// TIA Portal V17 export
// export: Created 2024-09-02T12:50:08.8547396Z, ExportSetting WithDefaults, DisplayName Totally Integrated Automation Portal, DisplayVersion V17, DisplayName TIA Portal Openness, DisplayVersion V17, DisplayName TIA Portal Version Control Interface, DisplayVersion V17, DisplayName STEP 7 Professional, DisplayVersion V17, DisplayName STEP 7 Safety, DisplayVersion V17, DisplayName WinCC Professional, DisplayVersion V17
FUNCTION "AnwFC2_FG02_Station_OP70" : Void   // FC1382, LAD
TITLE = Station
{ S7_Optimized_Access := 'TRUE' }
AUTHOR : VAF
FAMILY : SK
NAME : SK
VERSION : 0.1
// stored: AutoNumber false, IsIECCheckEnabled false, SetENOAutomatically false, UDAEnableTagReadback false
   VAR_TEMP
      Motion_Release : Bool;   // Motion permit
      Hand : Bool;
      Auto : Bool;
      t_Ret_Val_SFC : Int;
      t_fm_Gen : Bool;
      t_ParityFault : Bool;
      t_ConfigFault : Bool;
      t_Retval : Bool;
      MM150_Work : Bool;
      MM150_Home : Bool;
      MM160_Work : Bool;
      MM160_Home : Bool;
      MM170_Work : Bool;
      MM170_Home : Bool;
      MM140_Home : Bool;
      MM140_Work : Bool;
      X1 : Int;
      X2 : Int;
      Y : Int;
      X_actual : Int;
      dummy : Bool;
   END_VAR
   VAR_TEMP   // added for the SCL form of the ladder/FBD networks
      _w1 : Bool;
      _w2 : Bool;
   END_VAR
BEGIN

REGION Network 1: Motion permit / Hand/ Auto
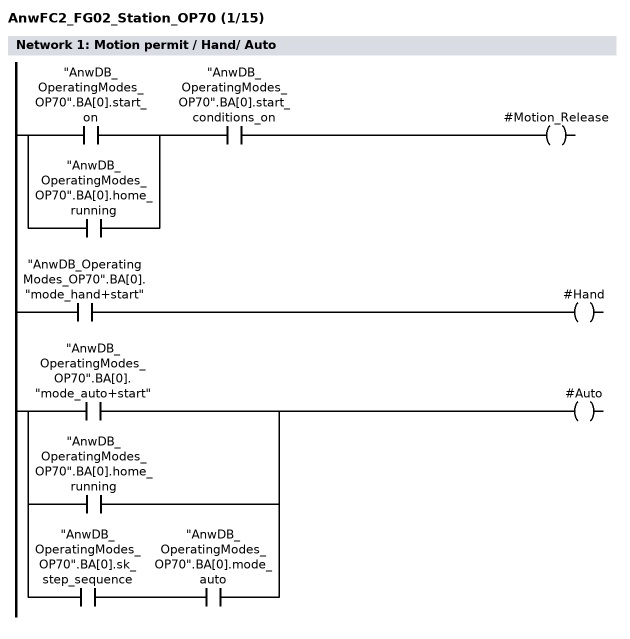
   RUNG wire#powerrail
      Contact( "AnwDB_OperatingModes_OP70".BA[0].start_on )
      wire#w1
      Contact( "AnwDB_OperatingModes_OP70".BA[0].start_conditions_on )
      Coil( #Motion_Release )
   END_RUNG
   RUNG wire#powerrail
      Contact( "AnwDB_OperatingModes_OP70".BA[0].home_running )
   END_RUNG wire#w1
   RUNG wire#powerrail
      Contact( "AnwDB_OperatingModes_OP70".BA[0]."mode_hand+start" )
      Coil( #Hand )
   END_RUNG
   RUNG wire#powerrail
      Contact( "AnwDB_OperatingModes_OP70".BA[0]."mode_auto+start" )
      wire#w2
      Coil( #Auto )
   END_RUNG
   RUNG wire#powerrail
      Contact( "AnwDB_OperatingModes_OP70".BA[0].home_running )
   END_RUNG wire#w2
   RUNG wire#powerrail
      Contact( "AnwDB_OperatingModes_OP70".BA[0].sk_step_sequence )
      Contact( "AnwDB_OperatingModes_OP70".BA[0].mode_auto )
   END_RUNG wire#w2
   // the same network as SCL:
   #Motion_Release := ("AnwDB_OperatingModes_OP70".BA[0].start_on OR "AnwDB_OperatingModes_OP70".BA[0].home_running) AND "AnwDB_OperatingModes_OP70".BA[0].start_conditions_on;
   #Hand := "AnwDB_OperatingModes_OP70".BA[0]."mode_hand+start";
   #Auto := "AnwDB_OperatingModes_OP70".BA[0]."mode_auto+start" OR "AnwDB_OperatingModes_OP70".BA[0].home_running OR ("AnwDB_OperatingModes_OP70".BA[0].sk_step_sequence AND "AnwDB_OperatingModes_OP70".BA[0].mode_auto);
END_REGION

REGION Network 2: Call of the step sequence
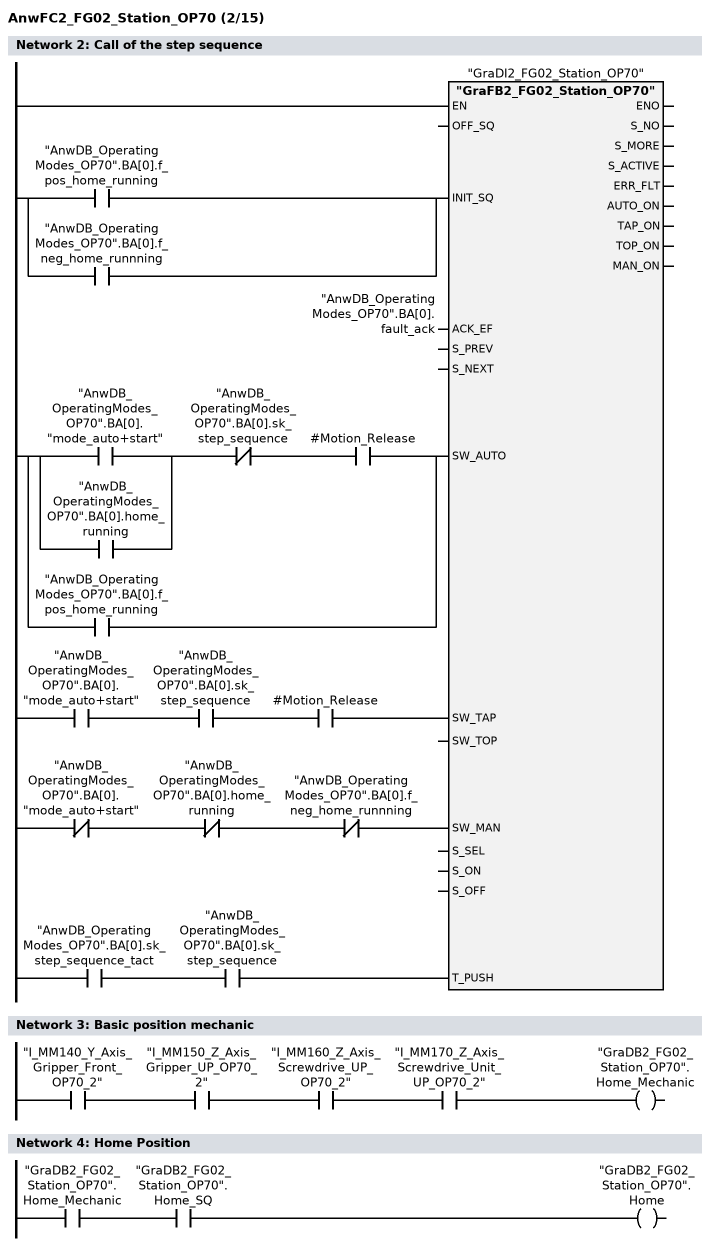
   RUNG wire#powerrail
      "GraDI2_FG02_Station_OP70"(INIT_SQ := wire#w1, SW_AUTO := wire#w3, SW_TAP := wire#w4, SW_MAN := wire#w5, T_PUSH := wire#w6, OFF_SQ :=, ACK_EF := "AnwDB_OperatingModes_OP70".BA[0].fault_ack, S_PREV :=, S_NEXT :=, SW_TOP :=, S_SEL :=, S_ON :=, S_OFF :=, S_NO =>, S_MORE =>, S_ACTIVE =>, ERR_FLT =>, AUTO_ON =>, TAP_ON =>, TOP_ON =>, MAN_ON =>)
   END_RUNG
   RUNG wire#powerrail
      Contact( "AnwDB_OperatingModes_OP70".BA[0].f_pos_home_running )
   END_RUNG wire#w1
   RUNG wire#powerrail
      Contact( "AnwDB_OperatingModes_OP70".BA[0].f_neg_home_runnning )
   END_RUNG wire#w1
   RUNG wire#powerrail
      Contact( "AnwDB_OperatingModes_OP70".BA[0]."mode_auto+start" )
      wire#w2
      I_Contact( "AnwDB_OperatingModes_OP70".BA[0].sk_step_sequence )
      Contact( #Motion_Release )
   END_RUNG wire#w3
   RUNG wire#powerrail
      Contact( "AnwDB_OperatingModes_OP70".BA[0].home_running )
   END_RUNG wire#w2
   RUNG wire#powerrail
      Contact( "AnwDB_OperatingModes_OP70".BA[0].f_pos_home_running )
   END_RUNG wire#w3
   RUNG wire#powerrail
      Contact( "AnwDB_OperatingModes_OP70".BA[0]."mode_auto+start" )
      Contact( "AnwDB_OperatingModes_OP70".BA[0].sk_step_sequence )
      Contact( #Motion_Release )
   END_RUNG wire#w4
   RUNG wire#powerrail
      I_Contact( "AnwDB_OperatingModes_OP70".BA[0]."mode_auto+start" )
      I_Contact( "AnwDB_OperatingModes_OP70".BA[0].home_running )
      I_Contact( "AnwDB_OperatingModes_OP70".BA[0].f_neg_home_runnning )
   END_RUNG wire#w5
   RUNG wire#powerrail
      Contact( "AnwDB_OperatingModes_OP70".BA[0].sk_step_sequence_tact )
      Contact( "AnwDB_OperatingModes_OP70".BA[0].sk_step_sequence )
   END_RUNG wire#w6
   // the same network as SCL:
   "GraDI2_FG02_Station_OP70"(INIT_SQ := "AnwDB_OperatingModes_OP70".BA[0].f_pos_home_running OR "AnwDB_OperatingModes_OP70".BA[0].f_neg_home_runnning,   // "GraFB2_FG02_Station_OP70"
                           ACK_EF := "AnwDB_OperatingModes_OP70".BA[0].fault_ack,
                           SW_AUTO := (("AnwDB_OperatingModes_OP70".BA[0]."mode_auto+start" OR "AnwDB_OperatingModes_OP70".BA[0].home_running) AND NOT "AnwDB_OperatingModes_OP70".BA[0].sk_step_sequence AND #Motion_Release) OR "AnwDB_OperatingModes_OP70".BA[0].f_pos_home_running,
                           SW_TAP := "AnwDB_OperatingModes_OP70".BA[0]."mode_auto+start" AND "AnwDB_OperatingModes_OP70".BA[0].sk_step_sequence AND #Motion_Release,
                           SW_MAN := NOT "AnwDB_OperatingModes_OP70".BA[0]."mode_auto+start" AND NOT "AnwDB_OperatingModes_OP70".BA[0].home_running AND NOT "AnwDB_OperatingModes_OP70".BA[0].f_neg_home_runnning,
                           T_PUSH := "AnwDB_OperatingModes_OP70".BA[0].sk_step_sequence_tact AND "AnwDB_OperatingModes_OP70".BA[0].sk_step_sequence);
END_REGION

REGION Network 3: Basic position mechanic
   RUNG wire#powerrail
      Contact( "I_MM140_Y_Axis_Gripper_Front_OP70_2" )
      Contact( "I_MM150_Z_Axis_Gripper_UP_OP70_2" )
      Contact( "I_MM160_Z_Axis_Screwdrive_UP_OP70_2" )
      Contact( "I_MM170_Z_Axis_Screwdrive_Unit_UP_OP70_2" )
      Coil( "GraDB2_FG02_Station_OP70".Home_Mechanic )
   END_RUNG
   // the same network as SCL:
   "GraDB2_FG02_Station_OP70".Home_Mechanic := "I_MM140_Y_Axis_Gripper_Front_OP70_2" AND "I_MM150_Z_Axis_Gripper_UP_OP70_2" AND "I_MM160_Z_Axis_Screwdrive_UP_OP70_2" AND "I_MM170_Z_Axis_Screwdrive_Unit_UP_OP70_2";
END_REGION

REGION Network 4: Home Position
   RUNG wire#powerrail
      Contact( "GraDB2_FG02_Station_OP70".Home_Mechanic )
      Contact( "GraDB2_FG02_Station_OP70".Home_SQ )
      Coil( "GraDB2_FG02_Station_OP70".Home )
   END_RUNG
   // the same network as SCL:
   "GraDB2_FG02_Station_OP70".Home := "GraDB2_FG02_Station_OP70".Home_Mechanic AND "GraDB2_FG02_Station_OP70".Home_SQ;
END_REGION

REGION Network 5: ########### USER ###########
END_REGION

REGION Network 6: Screen selection with NOK BEA1
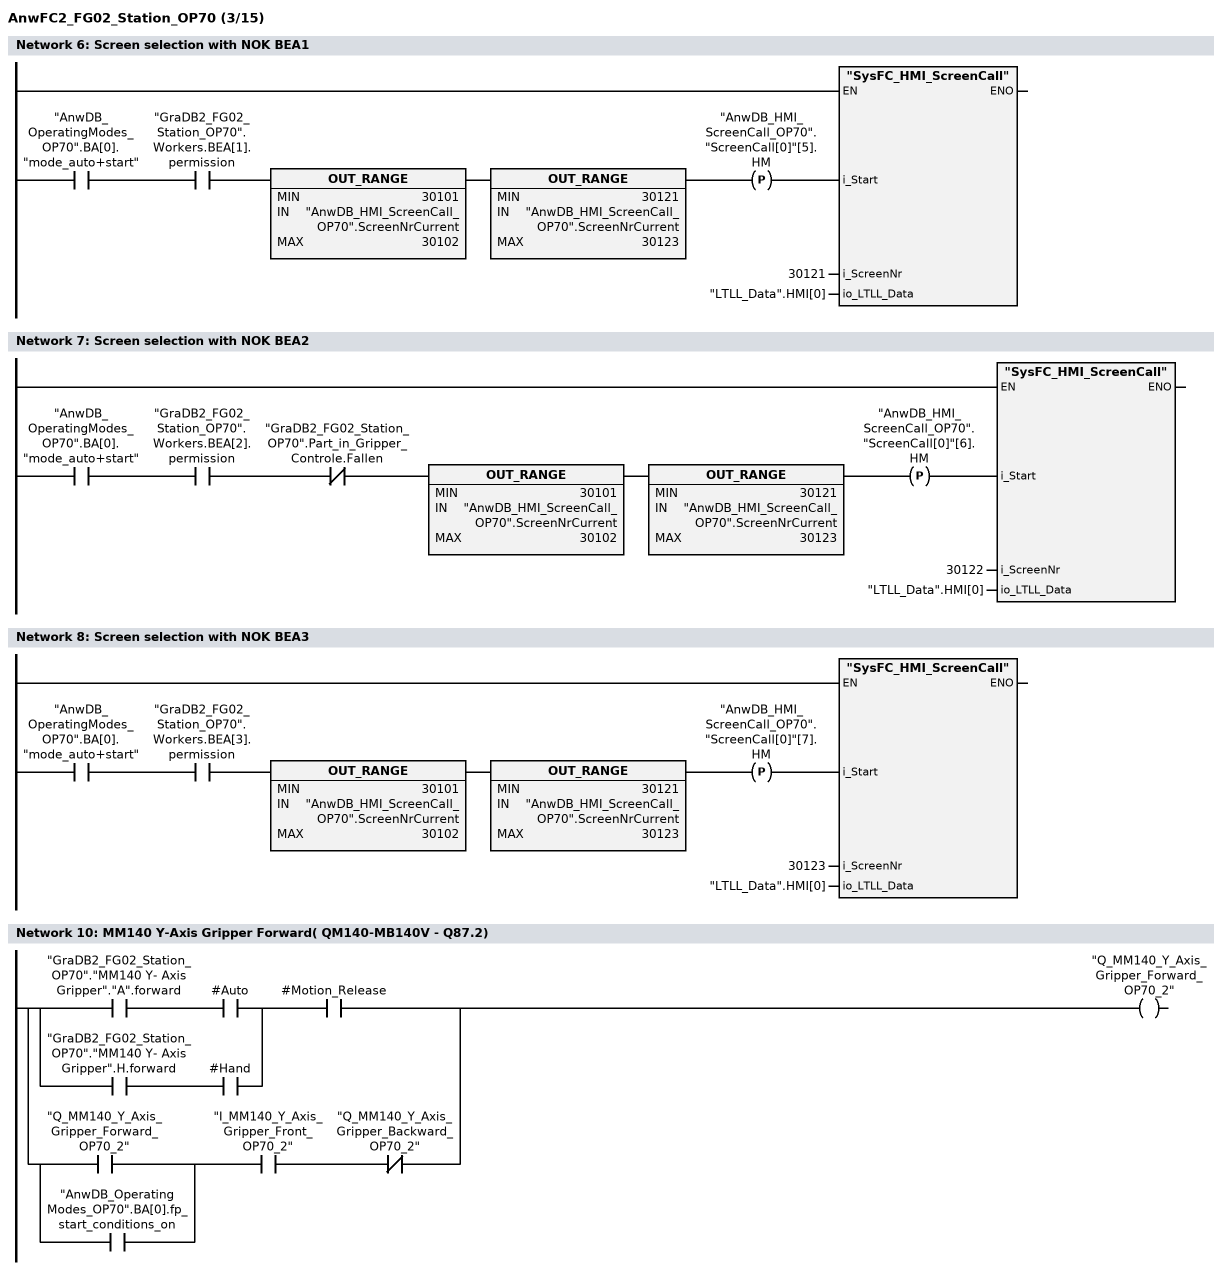
   #_w1 := "AnwDB_OperatingModes_OP70".BA[0]."mode_auto+start" AND "GraDB2_FG02_Station_OP70".Workers.BEA[1].permission AND (("AnwDB_HMI_ScreenCall_OP70".ScreenNrCurrent < 30101) OR ("AnwDB_HMI_ScreenCall_OP70".ScreenNrCurrent > 30102)) AND (("AnwDB_HMI_ScreenCall_OP70".ScreenNrCurrent < 30121) OR ("AnwDB_HMI_ScreenCall_OP70".ScreenNrCurrent > 30123));
   #_w2 := #_w1 AND NOT "AnwDB_HMI_ScreenCall_OP70"."ScreenCall[0]"[5].HM;   // rising edge
   "AnwDB_HMI_ScreenCall_OP70"."ScreenCall[0]"[5].HM := #_w1;
   "SysFC_HMI_ScreenCall"(i_Start := #_w2, i_ScreenNr := 30121, io_LTLL_Data := "LTLL_Data".HMI[0]);
END_REGION

REGION Network 7: Screen selection with NOK BEA2
   #_w1 := "AnwDB_OperatingModes_OP70".BA[0]."mode_auto+start" AND "GraDB2_FG02_Station_OP70".Workers.BEA[2].permission AND NOT "GraDB2_FG02_Station_OP70".Part_in_Gripper_Controle.Fallen AND (("AnwDB_HMI_ScreenCall_OP70".ScreenNrCurrent < 30101) OR ("AnwDB_HMI_ScreenCall_OP70".ScreenNrCurrent > 30102)) AND (("AnwDB_HMI_ScreenCall_OP70".ScreenNrCurrent < 30121) OR ("AnwDB_HMI_ScreenCall_OP70".ScreenNrCurrent > 30123));
   #_w2 := #_w1 AND NOT "AnwDB_HMI_ScreenCall_OP70"."ScreenCall[0]"[6].HM;   // rising edge
   "AnwDB_HMI_ScreenCall_OP70"."ScreenCall[0]"[6].HM := #_w1;
   "SysFC_HMI_ScreenCall"(i_Start := #_w2, i_ScreenNr := 30122, io_LTLL_Data := "LTLL_Data".HMI[0]);
END_REGION

REGION Network 8: Screen selection with NOK BEA3
   #_w1 := "AnwDB_OperatingModes_OP70".BA[0]."mode_auto+start" AND "GraDB2_FG02_Station_OP70".Workers.BEA[3].permission AND (("AnwDB_HMI_ScreenCall_OP70".ScreenNrCurrent < 30101) OR ("AnwDB_HMI_ScreenCall_OP70".ScreenNrCurrent > 30102)) AND (("AnwDB_HMI_ScreenCall_OP70".ScreenNrCurrent < 30121) OR ("AnwDB_HMI_ScreenCall_OP70".ScreenNrCurrent > 30123));
   #_w2 := #_w1 AND NOT "AnwDB_HMI_ScreenCall_OP70"."ScreenCall[0]"[7].HM;   // rising edge
   "AnwDB_HMI_ScreenCall_OP70"."ScreenCall[0]"[7].HM := #_w1;
   "SysFC_HMI_ScreenCall"(i_Start := #_w2, i_ScreenNr := 30123, io_LTLL_Data := "LTLL_Data".HMI[0]);
END_REGION

REGION Network 9: ########### SS_02_001_Setup ###########
END_REGION

REGION Network 10: MM140 Y-Axis Gripper Forward( QM140-MB140V - Q87.2)
   RUNG wire#powerrail
      Contact( "GraDB2_FG02_Station_OP70"."MM140 Y- Axis Gripper"."A".forward )
      Contact( #Auto )
      wire#w1
      Contact( #Motion_Release )
      wire#w2
      Coil( "Q_MM140_Y_Axis_Gripper_Forward_OP70_2" )
   END_RUNG
   RUNG wire#powerrail
      Contact( "GraDB2_FG02_Station_OP70"."MM140 Y- Axis Gripper".H.forward )
      Contact( #Hand )
   END_RUNG wire#w1
   RUNG wire#powerrail
      Contact( "Q_MM140_Y_Axis_Gripper_Forward_OP70_2" )
      wire#w3
      Contact( "I_MM140_Y_Axis_Gripper_Front_OP70_2" )
      I_Contact( "Q_MM140_Y_Axis_Gripper_Backward_OP70_2" )
   END_RUNG wire#w2
   RUNG wire#powerrail
      Contact( "AnwDB_OperatingModes_OP70".BA[0].fp_start_conditions_on )
   END_RUNG wire#w3
   // the same network as SCL:
   "Q_MM140_Y_Axis_Gripper_Forward_OP70_2" := ((("GraDB2_FG02_Station_OP70"."MM140 Y- Axis Gripper"."A".forward AND #Auto) OR ("GraDB2_FG02_Station_OP70"."MM140 Y- Axis Gripper".H.forward AND #Hand)) AND #Motion_Release) OR (("Q_MM140_Y_Axis_Gripper_Forward_OP70_2" OR "AnwDB_OperatingModes_OP70".BA[0].fp_start_conditions_on) AND "I_MM140_Y_Axis_Gripper_Front_OP70_2" AND NOT "Q_MM140_Y_Axis_Gripper_Backward_OP70_2");
END_REGION

REGION Network 11: MM140 Y-Axis Gripper Backward( QM140-MB140R - Q87.3 )
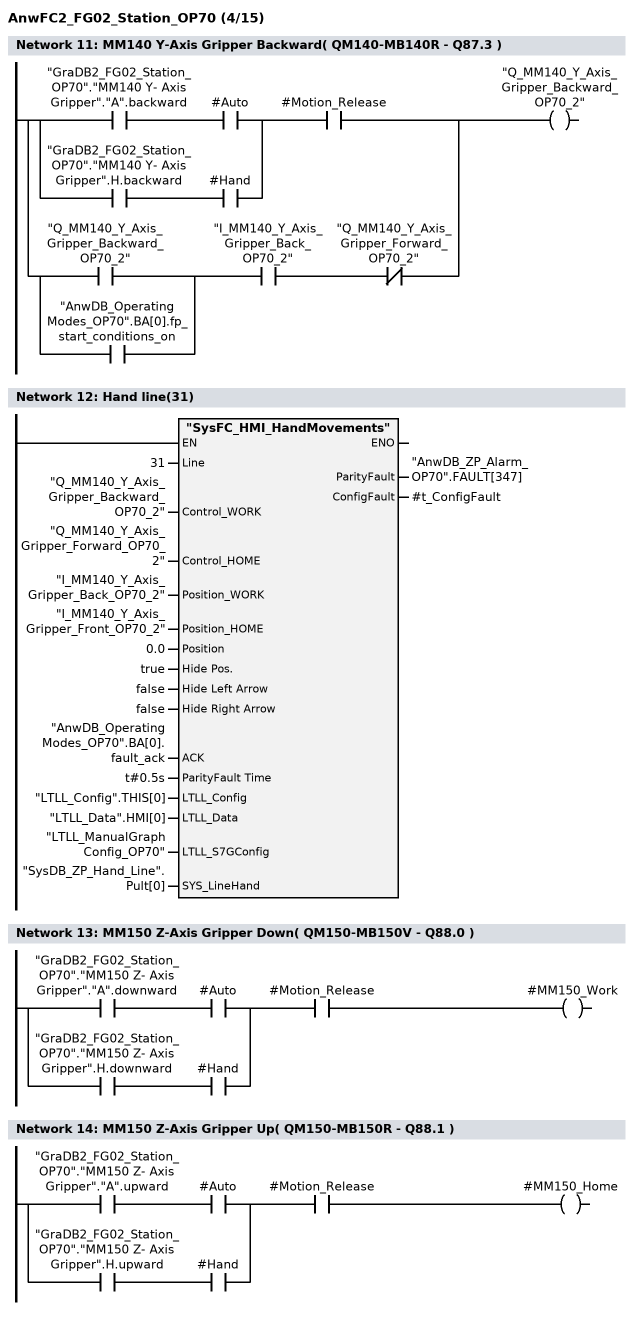
   RUNG wire#powerrail
      Contact( "GraDB2_FG02_Station_OP70"."MM140 Y- Axis Gripper"."A".backward )
      Contact( #Auto )
      wire#w1
      Contact( #Motion_Release )
      wire#w2
      Coil( "Q_MM140_Y_Axis_Gripper_Backward_OP70_2" )
   END_RUNG
   RUNG wire#powerrail
      Contact( "GraDB2_FG02_Station_OP70"."MM140 Y- Axis Gripper".H.backward )
      Contact( #Hand )
   END_RUNG wire#w1
   RUNG wire#powerrail
      Contact( "Q_MM140_Y_Axis_Gripper_Backward_OP70_2" )
      wire#w3
      Contact( "I_MM140_Y_Axis_Gripper_Back_OP70_2" )
      I_Contact( "Q_MM140_Y_Axis_Gripper_Forward_OP70_2" )
   END_RUNG wire#w2
   RUNG wire#powerrail
      Contact( "AnwDB_OperatingModes_OP70".BA[0].fp_start_conditions_on )
   END_RUNG wire#w3
   // the same network as SCL:
   "Q_MM140_Y_Axis_Gripper_Backward_OP70_2" := ((("GraDB2_FG02_Station_OP70"."MM140 Y- Axis Gripper"."A".backward AND #Auto) OR ("GraDB2_FG02_Station_OP70"."MM140 Y- Axis Gripper".H.backward AND #Hand)) AND #Motion_Release) OR (("Q_MM140_Y_Axis_Gripper_Backward_OP70_2" OR "AnwDB_OperatingModes_OP70".BA[0].fp_start_conditions_on) AND "I_MM140_Y_Axis_Gripper_Back_OP70_2" AND NOT "Q_MM140_Y_Axis_Gripper_Forward_OP70_2");
END_REGION

REGION Network 12: Hand line(31)
   RUNG wire#powerrail
      "SysFC_HMI_HandMovements"(Line := 31, Control_WORK := "Q_MM140_Y_Axis_Gripper_Backward_OP70_2", Control_HOME := "Q_MM140_Y_Axis_Gripper_Forward_OP70_2", Position_WORK := "I_MM140_Y_Axis_Gripper_Back_OP70_2", Position_HOME := "I_MM140_Y_Axis_Gripper_Front_OP70_2", Position := 0.0, "Hide Pos." := true, "Hide Left Arrow" := false, "Hide Right Arrow" := false, ACK := "AnwDB_OperatingModes_OP70".BA[0].fault_ack, "ParityFault Time" := t#0.5s, LTLL_Config := "LTLL_Config".THIS[0], LTLL_Data := "LTLL_Data".HMI[0], LTLL_S7GConfig := "LTLL_ManualGraphConfig_OP70", SYS_LineHand := "SysDB_ZP_Hand_Line".Pult[0], ParityFault => "AnwDB_ZP_Alarm_OP70".FAULT[347], ConfigFault => #t_ConfigFault)
   END_RUNG
   // the same network as SCL:
   "SysFC_HMI_HandMovements"(Line := 31,
                           Control_WORK := "Q_MM140_Y_Axis_Gripper_Backward_OP70_2",
                           Control_HOME := "Q_MM140_Y_Axis_Gripper_Forward_OP70_2",
                           Position_WORK := "I_MM140_Y_Axis_Gripper_Back_OP70_2",
                           Position_HOME := "I_MM140_Y_Axis_Gripper_Front_OP70_2",
                           Position := 0.0,
                           "Hide Pos." := true,
                           "Hide Left Arrow" := false,
                           "Hide Right Arrow" := false,
                           ACK := "AnwDB_OperatingModes_OP70".BA[0].fault_ack,
                           "ParityFault Time" := t#0.5s,
                           LTLL_Config := "LTLL_Config".THIS[0],
                           LTLL_Data := "LTLL_Data".HMI[0],
                           LTLL_S7GConfig := "LTLL_ManualGraphConfig_OP70",
                           SYS_LineHand := "SysDB_ZP_Hand_Line".Pult[0],
                           ParityFault => "AnwDB_ZP_Alarm_OP70".FAULT[347],
                           ConfigFault => #t_ConfigFault);
END_REGION

REGION Network 13: MM150 Z-Axis Gripper Down( QM150-MB150V - Q88.0 )
   RUNG wire#powerrail
      Contact( "GraDB2_FG02_Station_OP70"."MM150 Z- Axis Gripper"."A".downward )
      Contact( #Auto )
      wire#w1
      Contact( #Motion_Release )
      Coil( #MM150_Work )
   END_RUNG
   RUNG wire#powerrail
      Contact( "GraDB2_FG02_Station_OP70"."MM150 Z- Axis Gripper".H.downward )
      Contact( #Hand )
   END_RUNG wire#w1
   // the same network as SCL:
   #MM150_Work := (("GraDB2_FG02_Station_OP70"."MM150 Z- Axis Gripper"."A".downward AND #Auto) OR ("GraDB2_FG02_Station_OP70"."MM150 Z- Axis Gripper".H.downward AND #Hand)) AND #Motion_Release;
END_REGION

REGION Network 14: MM150 Z-Axis Gripper Up( QM150-MB150R - Q88.1 )
   RUNG wire#powerrail
      Contact( "GraDB2_FG02_Station_OP70"."MM150 Z- Axis Gripper"."A".upward )
      Contact( #Auto )
      wire#w1
      Contact( #Motion_Release )
      Coil( #MM150_Home )
   END_RUNG
   RUNG wire#powerrail
      Contact( "GraDB2_FG02_Station_OP70"."MM150 Z- Axis Gripper".H.upward )
      Contact( #Hand )
   END_RUNG wire#w1
   // the same network as SCL:
   #MM150_Home := (("GraDB2_FG02_Station_OP70"."MM150 Z- Axis Gripper"."A".upward AND #Auto) OR ("GraDB2_FG02_Station_OP70"."MM150 Z- Axis Gripper".H.upward AND #Hand)) AND #Motion_Release;
END_REGION

REGION Network 15: HLP - Z-Axis Gripper Up/Down
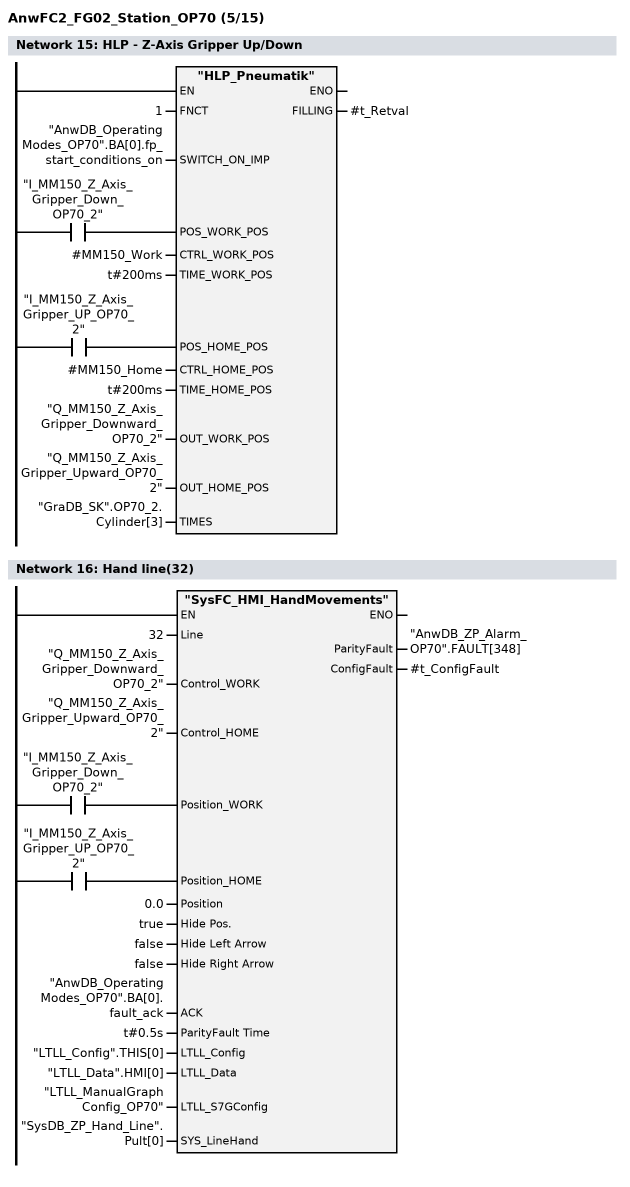
   RUNG wire#powerrail
      "HLP_Pneumatik"(POS_WORK_POS := wire#w1, POS_HOME_POS := wire#w2, FNCT := 1, SWITCH_ON_IMP := "AnwDB_OperatingModes_OP70".BA[0].fp_start_conditions_on, CTRL_WORK_POS := #MM150_Work, TIME_WORK_POS := t#200ms, CTRL_HOME_POS := #MM150_Home, TIME_HOME_POS := t#200ms, OUT_WORK_POS := "Q_MM150_Z_Axis_Gripper_Downward_OP70_2", OUT_HOME_POS := "Q_MM150_Z_Axis_Gripper_Upward_OP70_2", TIMES := "GraDB_SK".OP70_2.Cylinder[3], FILLING => #t_Retval)
   END_RUNG
   RUNG wire#powerrail
      Contact( "I_MM150_Z_Axis_Gripper_Down_OP70_2" )
   END_RUNG wire#w1
   RUNG wire#powerrail
      Contact( "I_MM150_Z_Axis_Gripper_UP_OP70_2" )
   END_RUNG wire#w2
   // the same network as SCL:
   "HLP_Pneumatik"(FNCT := 1,
                   SWITCH_ON_IMP := "AnwDB_OperatingModes_OP70".BA[0].fp_start_conditions_on,
                   POS_WORK_POS := "I_MM150_Z_Axis_Gripper_Down_OP70_2",
                   CTRL_WORK_POS := #MM150_Work,
                   TIME_WORK_POS := t#200ms,
                   POS_HOME_POS := "I_MM150_Z_Axis_Gripper_UP_OP70_2",
                   CTRL_HOME_POS := #MM150_Home,
                   TIME_HOME_POS := t#200ms,
                   OUT_WORK_POS := "Q_MM150_Z_Axis_Gripper_Downward_OP70_2",
                   OUT_HOME_POS := "Q_MM150_Z_Axis_Gripper_Upward_OP70_2",
                   TIMES := "GraDB_SK".OP70_2.Cylinder[3],
                   FILLING => #t_Retval);
END_REGION

REGION Network 16: Hand line(32)
   RUNG wire#powerrail
      "SysFC_HMI_HandMovements"(Position_WORK := wire#w1, Position_HOME := wire#w2, Line := 32, Control_WORK := "Q_MM150_Z_Axis_Gripper_Downward_OP70_2", Control_HOME := "Q_MM150_Z_Axis_Gripper_Upward_OP70_2", Position := 0.0, "Hide Pos." := true, "Hide Left Arrow" := false, "Hide Right Arrow" := false, ACK := "AnwDB_OperatingModes_OP70".BA[0].fault_ack, "ParityFault Time" := t#0.5s, LTLL_Config := "LTLL_Config".THIS[0], LTLL_Data := "LTLL_Data".HMI[0], LTLL_S7GConfig := "LTLL_ManualGraphConfig_OP70", SYS_LineHand := "SysDB_ZP_Hand_Line".Pult[0], ParityFault => "AnwDB_ZP_Alarm_OP70".FAULT[348], ConfigFault => #t_ConfigFault)
   END_RUNG
   RUNG wire#powerrail
      Contact( "I_MM150_Z_Axis_Gripper_Down_OP70_2" )
   END_RUNG wire#w1
   RUNG wire#powerrail
      Contact( "I_MM150_Z_Axis_Gripper_UP_OP70_2" )
   END_RUNG wire#w2
   // the same network as SCL:
   "SysFC_HMI_HandMovements"(Line := 32,
                           Control_WORK := "Q_MM150_Z_Axis_Gripper_Downward_OP70_2",
                           Control_HOME := "Q_MM150_Z_Axis_Gripper_Upward_OP70_2",
                           Position_WORK := "I_MM150_Z_Axis_Gripper_Down_OP70_2",
                           Position_HOME := "I_MM150_Z_Axis_Gripper_UP_OP70_2",
                           Position := 0.0,
                           "Hide Pos." := true,
                           "Hide Left Arrow" := false,
                           "Hide Right Arrow" := false,
                           ACK := "AnwDB_OperatingModes_OP70".BA[0].fault_ack,
                           "ParityFault Time" := t#0.5s,
                           LTLL_Config := "LTLL_Config".THIS[0],
                           LTLL_Data := "LTLL_Data".HMI[0],
                           LTLL_S7GConfig := "LTLL_ManualGraphConfig_OP70",
                           SYS_LineHand := "SysDB_ZP_Hand_Line".Pult[0],
                           ParityFault => "AnwDB_ZP_Alarm_OP70".FAULT[348],
                           ConfigFault => #t_ConfigFault);
END_REGION

REGION Network 17: Voccum Gripper Open ######( QM303-MBXXXR - Q2.1)
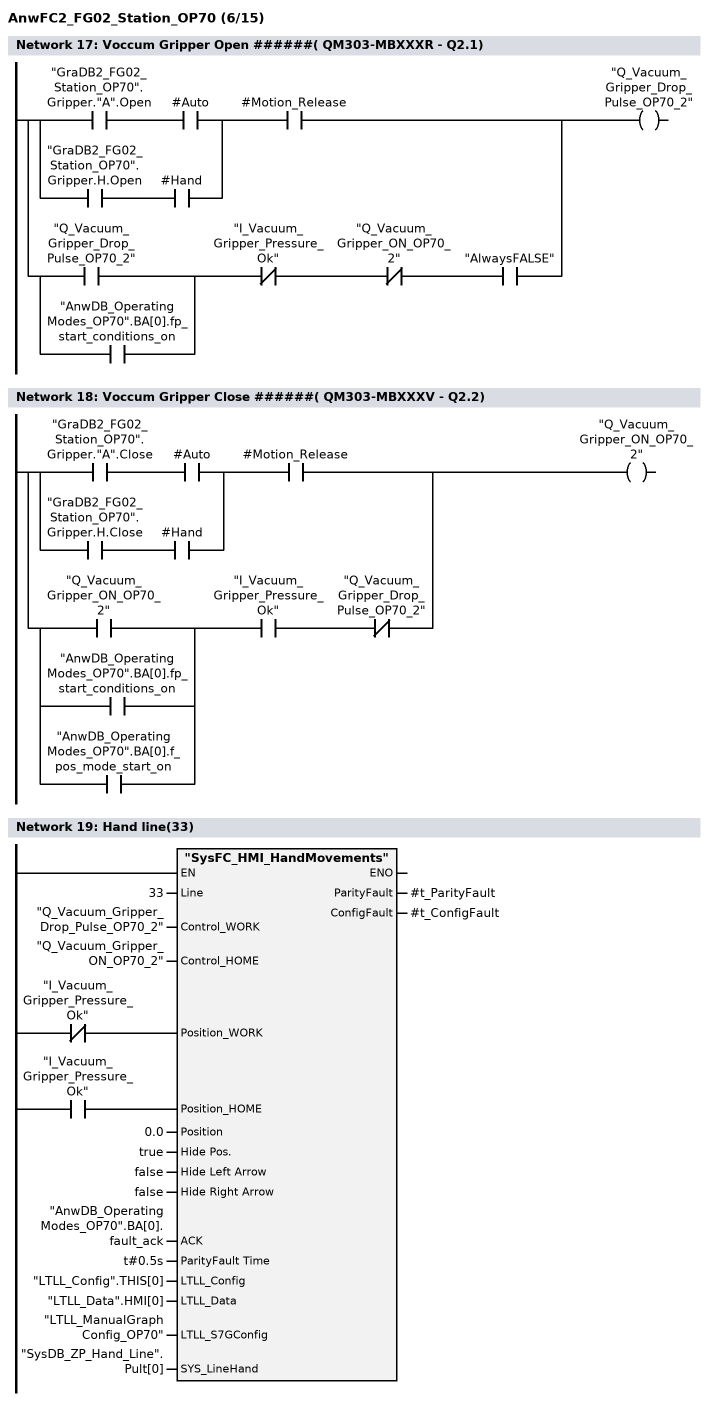
   RUNG wire#powerrail
      Contact( "GraDB2_FG02_Station_OP70".Gripper."A".Open )
      Contact( #Auto )
      wire#w1
      Contact( #Motion_Release )
      wire#w2
      Coil( "Q_Vacuum_Gripper_Drop_Pulse_OP70_2" )
   END_RUNG
   RUNG wire#powerrail
      Contact( "GraDB2_FG02_Station_OP70".Gripper.H.Open )
      Contact( #Hand )
   END_RUNG wire#w1
   RUNG wire#powerrail
      Contact( "Q_Vacuum_Gripper_Drop_Pulse_OP70_2" )
      wire#w3
      I_Contact( "I_Vacuum_Gripper_Pressure_Ok" )
      I_Contact( "Q_Vacuum_Gripper_ON_OP70_2" )
      Contact( "AlwaysFALSE" )
   END_RUNG wire#w2
   RUNG wire#powerrail
      Contact( "AnwDB_OperatingModes_OP70".BA[0].fp_start_conditions_on )
   END_RUNG wire#w3
   // the same network as SCL:
   "Q_Vacuum_Gripper_Drop_Pulse_OP70_2" := ((("GraDB2_FG02_Station_OP70".Gripper."A".Open AND #Auto) OR ("GraDB2_FG02_Station_OP70".Gripper.H.Open AND #Hand)) AND #Motion_Release) OR (("Q_Vacuum_Gripper_Drop_Pulse_OP70_2" OR "AnwDB_OperatingModes_OP70".BA[0].fp_start_conditions_on) AND NOT "I_Vacuum_Gripper_Pressure_Ok" AND NOT "Q_Vacuum_Gripper_ON_OP70_2" AND "AlwaysFALSE");
END_REGION

REGION Network 18: Voccum Gripper Close ######( QM303-MBXXXV - Q2.2)
   RUNG wire#powerrail
      Contact( "GraDB2_FG02_Station_OP70".Gripper."A".Close )
      Contact( #Auto )
      wire#w1
      Contact( #Motion_Release )
      wire#w2
      Coil( "Q_Vacuum_Gripper_ON_OP70_2" )
   END_RUNG
   RUNG wire#powerrail
      Contact( "GraDB2_FG02_Station_OP70".Gripper.H.Close )
      Contact( #Hand )
   END_RUNG wire#w1
   RUNG wire#powerrail
      Contact( "Q_Vacuum_Gripper_ON_OP70_2" )
      wire#w3
      Contact( "I_Vacuum_Gripper_Pressure_Ok" )
      I_Contact( "Q_Vacuum_Gripper_Drop_Pulse_OP70_2" )
   END_RUNG wire#w2
   RUNG wire#powerrail
      Contact( "AnwDB_OperatingModes_OP70".BA[0].fp_start_conditions_on )
   END_RUNG wire#w3
   RUNG wire#powerrail
      Contact( "AnwDB_OperatingModes_OP70".BA[0].f_pos_mode_start_on )
   END_RUNG wire#w3
   // the same network as SCL:
   "Q_Vacuum_Gripper_ON_OP70_2" := ((("GraDB2_FG02_Station_OP70".Gripper."A".Close AND #Auto) OR ("GraDB2_FG02_Station_OP70".Gripper.H.Close AND #Hand)) AND #Motion_Release) OR (("Q_Vacuum_Gripper_ON_OP70_2" OR "AnwDB_OperatingModes_OP70".BA[0].fp_start_conditions_on OR "AnwDB_OperatingModes_OP70".BA[0].f_pos_mode_start_on) AND "I_Vacuum_Gripper_Pressure_Ok" AND NOT "Q_Vacuum_Gripper_Drop_Pulse_OP70_2");
END_REGION

REGION Network 19: Hand line(33)
   RUNG wire#powerrail
      "SysFC_HMI_HandMovements"(Position_WORK := wire#w1, Position_HOME := wire#w2, Line := 33, Control_WORK := "Q_Vacuum_Gripper_Drop_Pulse_OP70_2", Control_HOME := "Q_Vacuum_Gripper_ON_OP70_2", Position := 0.0, "Hide Pos." := true, "Hide Left Arrow" := false, "Hide Right Arrow" := false, ACK := "AnwDB_OperatingModes_OP70".BA[0].fault_ack, "ParityFault Time" := t#0.5s, LTLL_Config := "LTLL_Config".THIS[0], LTLL_Data := "LTLL_Data".HMI[0], LTLL_S7GConfig := "LTLL_ManualGraphConfig_OP70", SYS_LineHand := "SysDB_ZP_Hand_Line".Pult[0], ParityFault => #t_ParityFault, ConfigFault => #t_ConfigFault)
   END_RUNG
   RUNG wire#powerrail
      I_Contact( "I_Vacuum_Gripper_Pressure_Ok" )
   END_RUNG wire#w1
   RUNG wire#powerrail
      Contact( "I_Vacuum_Gripper_Pressure_Ok" )
   END_RUNG wire#w2
   // the same network as SCL:
   "SysFC_HMI_HandMovements"(Line := 33,
                           Control_WORK := "Q_Vacuum_Gripper_Drop_Pulse_OP70_2",
                           Control_HOME := "Q_Vacuum_Gripper_ON_OP70_2",
                           Position_WORK := NOT "I_Vacuum_Gripper_Pressure_Ok",
                           Position_HOME := "I_Vacuum_Gripper_Pressure_Ok",
                           Position := 0.0,
                           "Hide Pos." := true,
                           "Hide Left Arrow" := false,
                           "Hide Right Arrow" := false,
                           ACK := "AnwDB_OperatingModes_OP70".BA[0].fault_ack,
                           "ParityFault Time" := t#0.5s,
                           LTLL_Config := "LTLL_Config".THIS[0],
                           LTLL_Data := "LTLL_Data".HMI[0],
                           LTLL_S7GConfig := "LTLL_ManualGraphConfig_OP70",
                           SYS_LineHand := "SysDB_ZP_Hand_Line".Pult[0],
                           ParityFault => #t_ParityFault,
                           ConfigFault => #t_ConfigFault);
END_REGION

REGION Network 20: MM160 Z-Axis Screwdriver Down( QM160-MB160V - Q88.2 )
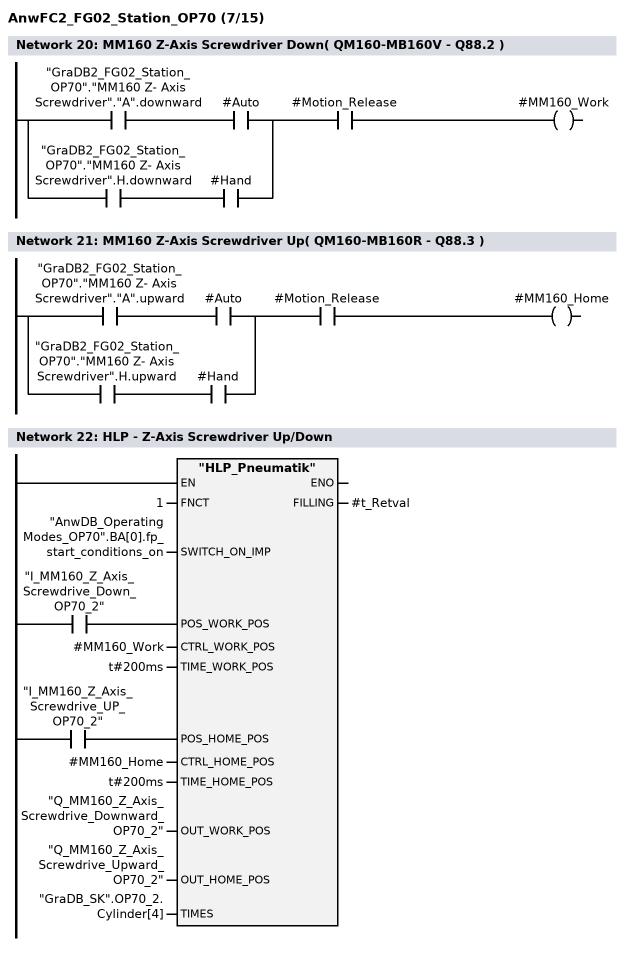
   RUNG wire#powerrail
      Contact( "GraDB2_FG02_Station_OP70"."MM160 Z- Axis Screwdriver"."A".downward )
      Contact( #Auto )
      wire#w1
      Contact( #Motion_Release )
      Coil( #MM160_Work )
   END_RUNG
   RUNG wire#powerrail
      Contact( "GraDB2_FG02_Station_OP70"."MM160 Z- Axis Screwdriver".H.downward )
      Contact( #Hand )
   END_RUNG wire#w1
   // the same network as SCL:
   #MM160_Work := (("GraDB2_FG02_Station_OP70"."MM160 Z- Axis Screwdriver"."A".downward AND #Auto) OR ("GraDB2_FG02_Station_OP70"."MM160 Z- Axis Screwdriver".H.downward AND #Hand)) AND #Motion_Release;
END_REGION

REGION Network 21: MM160 Z-Axis Screwdriver Up( QM160-MB160R - Q88.3 )
   RUNG wire#powerrail
      Contact( "GraDB2_FG02_Station_OP70"."MM160 Z- Axis Screwdriver"."A".upward )
      Contact( #Auto )
      wire#w1
      Contact( #Motion_Release )
      Coil( #MM160_Home )
   END_RUNG
   RUNG wire#powerrail
      Contact( "GraDB2_FG02_Station_OP70"."MM160 Z- Axis Screwdriver".H.upward )
      Contact( #Hand )
   END_RUNG wire#w1
   // the same network as SCL:
   #MM160_Home := (("GraDB2_FG02_Station_OP70"."MM160 Z- Axis Screwdriver"."A".upward AND #Auto) OR ("GraDB2_FG02_Station_OP70"."MM160 Z- Axis Screwdriver".H.upward AND #Hand)) AND #Motion_Release;
END_REGION

REGION Network 22: HLP - Z-Axis Screwdriver Up/Down
   RUNG wire#powerrail
      "HLP_Pneumatik"(POS_WORK_POS := wire#w1, POS_HOME_POS := wire#w2, FNCT := 1, SWITCH_ON_IMP := "AnwDB_OperatingModes_OP70".BA[0].fp_start_conditions_on, CTRL_WORK_POS := #MM160_Work, TIME_WORK_POS := t#200ms, CTRL_HOME_POS := #MM160_Home, TIME_HOME_POS := t#200ms, OUT_WORK_POS := "Q_MM160_Z_Axis_Screwdrive_Downward_OP70_2", OUT_HOME_POS := "Q_MM160_Z_Axis_Screwdrive_Upward_OP70_2", TIMES := "GraDB_SK".OP70_2.Cylinder[4], FILLING => #t_Retval)
   END_RUNG
   RUNG wire#powerrail
      Contact( "I_MM160_Z_Axis_Screwdrive_Down_OP70_2" )
   END_RUNG wire#w1
   RUNG wire#powerrail
      Contact( "I_MM160_Z_Axis_Screwdrive_UP_OP70_2" )
   END_RUNG wire#w2
   // the same network as SCL:
   "HLP_Pneumatik"(FNCT := 1,
                   SWITCH_ON_IMP := "AnwDB_OperatingModes_OP70".BA[0].fp_start_conditions_on,
                   POS_WORK_POS := "I_MM160_Z_Axis_Screwdrive_Down_OP70_2",
                   CTRL_WORK_POS := #MM160_Work,
                   TIME_WORK_POS := t#200ms,
                   POS_HOME_POS := "I_MM160_Z_Axis_Screwdrive_UP_OP70_2",
                   CTRL_HOME_POS := #MM160_Home,
                   TIME_HOME_POS := t#200ms,
                   OUT_WORK_POS := "Q_MM160_Z_Axis_Screwdrive_Downward_OP70_2",
                   OUT_HOME_POS := "Q_MM160_Z_Axis_Screwdrive_Upward_OP70_2",
                   TIMES := "GraDB_SK".OP70_2.Cylinder[4],
                   FILLING => #t_Retval);
END_REGION

REGION Network 23: Hand line(34)
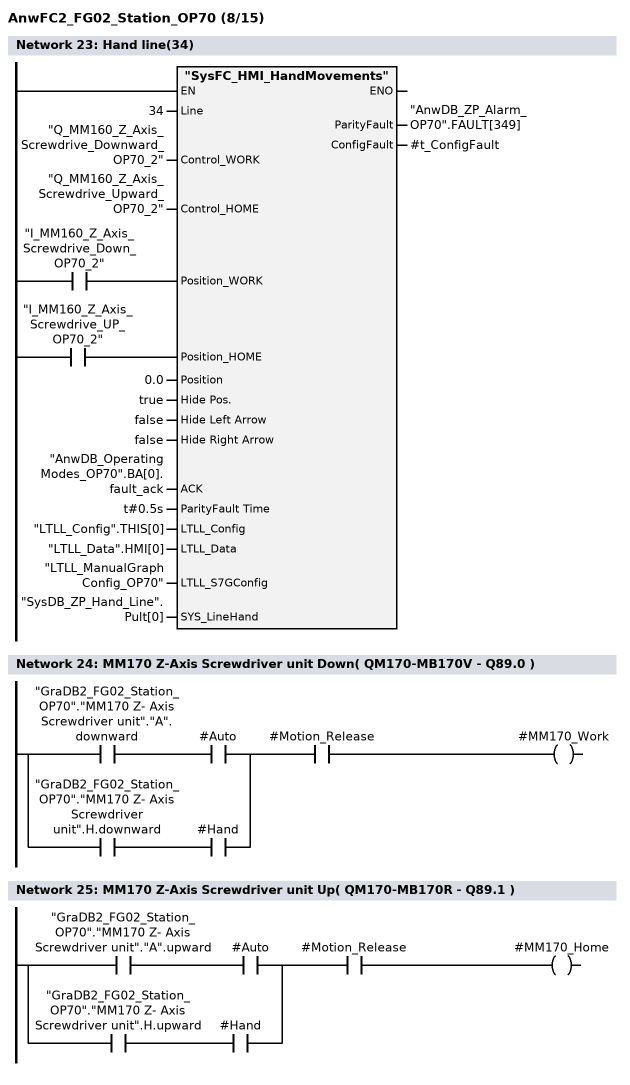
   RUNG wire#powerrail
      "SysFC_HMI_HandMovements"(Position_WORK := wire#w1, Position_HOME := wire#w2, Line := 34, Control_WORK := "Q_MM160_Z_Axis_Screwdrive_Downward_OP70_2", Control_HOME := "Q_MM160_Z_Axis_Screwdrive_Upward_OP70_2", Position := 0.0, "Hide Pos." := true, "Hide Left Arrow" := false, "Hide Right Arrow" := false, ACK := "AnwDB_OperatingModes_OP70".BA[0].fault_ack, "ParityFault Time" := t#0.5s, LTLL_Config := "LTLL_Config".THIS[0], LTLL_Data := "LTLL_Data".HMI[0], LTLL_S7GConfig := "LTLL_ManualGraphConfig_OP70", SYS_LineHand := "SysDB_ZP_Hand_Line".Pult[0], ParityFault => "AnwDB_ZP_Alarm_OP70".FAULT[349], ConfigFault => #t_ConfigFault)
   END_RUNG
   RUNG wire#powerrail
      Contact( "I_MM160_Z_Axis_Screwdrive_Down_OP70_2" )
   END_RUNG wire#w1
   RUNG wire#powerrail
      Contact( "I_MM160_Z_Axis_Screwdrive_UP_OP70_2" )
   END_RUNG wire#w2
   // the same network as SCL:
   "SysFC_HMI_HandMovements"(Line := 34,
                           Control_WORK := "Q_MM160_Z_Axis_Screwdrive_Downward_OP70_2",
                           Control_HOME := "Q_MM160_Z_Axis_Screwdrive_Upward_OP70_2",
                           Position_WORK := "I_MM160_Z_Axis_Screwdrive_Down_OP70_2",
                           Position_HOME := "I_MM160_Z_Axis_Screwdrive_UP_OP70_2",
                           Position := 0.0,
                           "Hide Pos." := true,
                           "Hide Left Arrow" := false,
                           "Hide Right Arrow" := false,
                           ACK := "AnwDB_OperatingModes_OP70".BA[0].fault_ack,
                           "ParityFault Time" := t#0.5s,
                           LTLL_Config := "LTLL_Config".THIS[0],
                           LTLL_Data := "LTLL_Data".HMI[0],
                           LTLL_S7GConfig := "LTLL_ManualGraphConfig_OP70",
                           SYS_LineHand := "SysDB_ZP_Hand_Line".Pult[0],
                           ParityFault => "AnwDB_ZP_Alarm_OP70".FAULT[349],
                           ConfigFault => #t_ConfigFault);
END_REGION

REGION Network 24: MM170 Z-Axis Screwdriver unit Down( QM170-MB170V - Q89.0 )
   RUNG wire#powerrail
      Contact( "GraDB2_FG02_Station_OP70"."MM170 Z- Axis Screwdriver unit"."A".downward )
      Contact( #Auto )
      wire#w1
      Contact( #Motion_Release )
      Coil( #MM170_Work )
   END_RUNG
   RUNG wire#powerrail
      Contact( "GraDB2_FG02_Station_OP70"."MM170 Z- Axis Screwdriver unit".H.downward )
      Contact( #Hand )
   END_RUNG wire#w1
   // the same network as SCL:
   #MM170_Work := (("GraDB2_FG02_Station_OP70"."MM170 Z- Axis Screwdriver unit"."A".downward AND #Auto) OR ("GraDB2_FG02_Station_OP70"."MM170 Z- Axis Screwdriver unit".H.downward AND #Hand)) AND #Motion_Release;
END_REGION

REGION Network 25: MM170 Z-Axis Screwdriver unit Up( QM170-MB170R - Q89.1 )
   RUNG wire#powerrail
      Contact( "GraDB2_FG02_Station_OP70"."MM170 Z- Axis Screwdriver unit"."A".upward )
      Contact( #Auto )
      wire#w1
      Contact( #Motion_Release )
      Coil( #MM170_Home )
   END_RUNG
   RUNG wire#powerrail
      Contact( "GraDB2_FG02_Station_OP70"."MM170 Z- Axis Screwdriver unit".H.upward )
      Contact( #Hand )
   END_RUNG wire#w1
   // the same network as SCL:
   #MM170_Home := (("GraDB2_FG02_Station_OP70"."MM170 Z- Axis Screwdriver unit"."A".upward AND #Auto) OR ("GraDB2_FG02_Station_OP70"."MM170 Z- Axis Screwdriver unit".H.upward AND #Hand)) AND #Motion_Release;
END_REGION

REGION Network 26: HLP - Z-Axis Screwdriver unit Up/Down
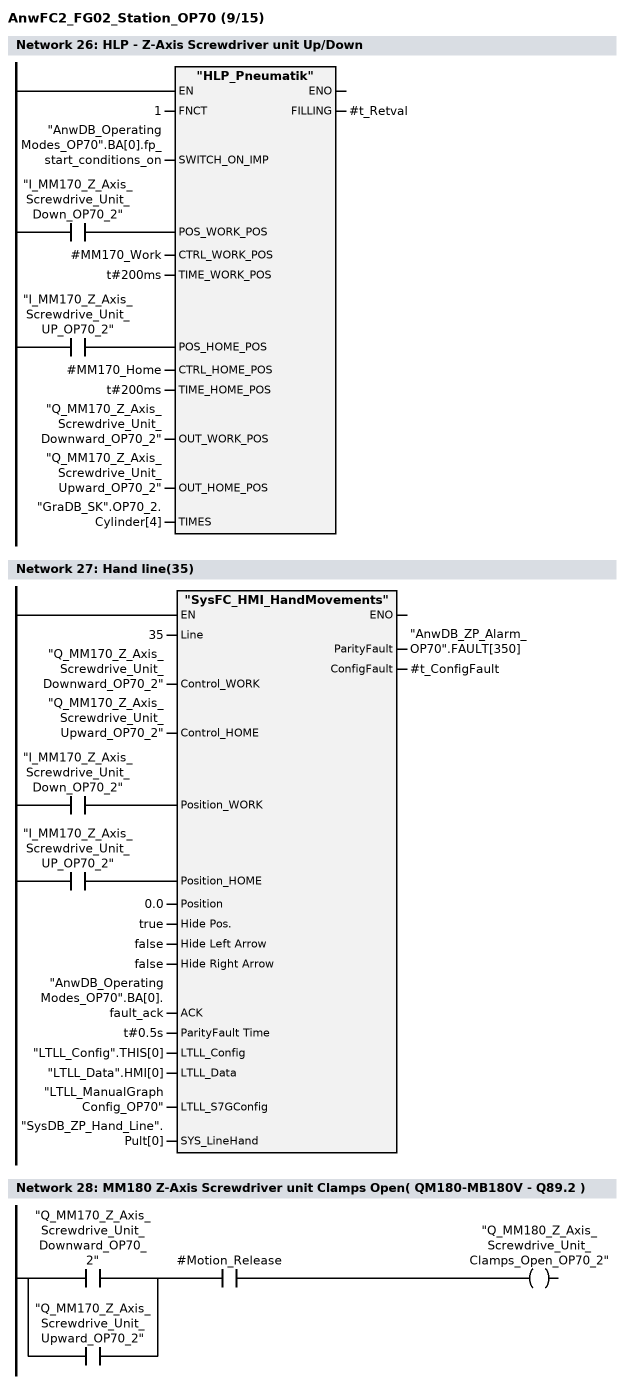
   RUNG wire#powerrail
      "HLP_Pneumatik"(POS_WORK_POS := wire#w1, POS_HOME_POS := wire#w2, FNCT := 1, SWITCH_ON_IMP := "AnwDB_OperatingModes_OP70".BA[0].fp_start_conditions_on, CTRL_WORK_POS := #MM170_Work, TIME_WORK_POS := t#200ms, CTRL_HOME_POS := #MM170_Home, TIME_HOME_POS := t#200ms, OUT_WORK_POS := "Q_MM170_Z_Axis_Screwdrive_Unit_Downward_OP70_2", OUT_HOME_POS := "Q_MM170_Z_Axis_Screwdrive_Unit_Upward_OP70_2", TIMES := "GraDB_SK".OP70_2.Cylinder[4], FILLING => #t_Retval)
   END_RUNG
   RUNG wire#powerrail
      Contact( "I_MM170_Z_Axis_Screwdrive_Unit_Down_OP70_2" )
   END_RUNG wire#w1
   RUNG wire#powerrail
      Contact( "I_MM170_Z_Axis_Screwdrive_Unit_UP_OP70_2" )
   END_RUNG wire#w2
   // the same network as SCL:
   "HLP_Pneumatik"(FNCT := 1,
                   SWITCH_ON_IMP := "AnwDB_OperatingModes_OP70".BA[0].fp_start_conditions_on,
                   POS_WORK_POS := "I_MM170_Z_Axis_Screwdrive_Unit_Down_OP70_2",
                   CTRL_WORK_POS := #MM170_Work,
                   TIME_WORK_POS := t#200ms,
                   POS_HOME_POS := "I_MM170_Z_Axis_Screwdrive_Unit_UP_OP70_2",
                   CTRL_HOME_POS := #MM170_Home,
                   TIME_HOME_POS := t#200ms,
                   OUT_WORK_POS := "Q_MM170_Z_Axis_Screwdrive_Unit_Downward_OP70_2",
                   OUT_HOME_POS := "Q_MM170_Z_Axis_Screwdrive_Unit_Upward_OP70_2",
                   TIMES := "GraDB_SK".OP70_2.Cylinder[4],
                   FILLING => #t_Retval);
END_REGION

REGION Network 27: Hand line(35)
   RUNG wire#powerrail
      "SysFC_HMI_HandMovements"(Position_WORK := wire#w1, Position_HOME := wire#w2, Line := 35, Control_WORK := "Q_MM170_Z_Axis_Screwdrive_Unit_Downward_OP70_2", Control_HOME := "Q_MM170_Z_Axis_Screwdrive_Unit_Upward_OP70_2", Position := 0.0, "Hide Pos." := true, "Hide Left Arrow" := false, "Hide Right Arrow" := false, ACK := "AnwDB_OperatingModes_OP70".BA[0].fault_ack, "ParityFault Time" := t#0.5s, LTLL_Config := "LTLL_Config".THIS[0], LTLL_Data := "LTLL_Data".HMI[0], LTLL_S7GConfig := "LTLL_ManualGraphConfig_OP70", SYS_LineHand := "SysDB_ZP_Hand_Line".Pult[0], ParityFault => "AnwDB_ZP_Alarm_OP70".FAULT[350], ConfigFault => #t_ConfigFault)
   END_RUNG
   RUNG wire#powerrail
      Contact( "I_MM170_Z_Axis_Screwdrive_Unit_Down_OP70_2" )
   END_RUNG wire#w1
   RUNG wire#powerrail
      Contact( "I_MM170_Z_Axis_Screwdrive_Unit_UP_OP70_2" )
   END_RUNG wire#w2
   // the same network as SCL:
   "SysFC_HMI_HandMovements"(Line := 35,
                           Control_WORK := "Q_MM170_Z_Axis_Screwdrive_Unit_Downward_OP70_2",
                           Control_HOME := "Q_MM170_Z_Axis_Screwdrive_Unit_Upward_OP70_2",
                           Position_WORK := "I_MM170_Z_Axis_Screwdrive_Unit_Down_OP70_2",
                           Position_HOME := "I_MM170_Z_Axis_Screwdrive_Unit_UP_OP70_2",
                           Position := 0.0,
                           "Hide Pos." := true,
                           "Hide Left Arrow" := false,
                           "Hide Right Arrow" := false,
                           ACK := "AnwDB_OperatingModes_OP70".BA[0].fault_ack,
                           "ParityFault Time" := t#0.5s,
                           LTLL_Config := "LTLL_Config".THIS[0],
                           LTLL_Data := "LTLL_Data".HMI[0],
                           LTLL_S7GConfig := "LTLL_ManualGraphConfig_OP70",
                           SYS_LineHand := "SysDB_ZP_Hand_Line".Pult[0],
                           ParityFault => "AnwDB_ZP_Alarm_OP70".FAULT[350],
                           ConfigFault => #t_ConfigFault);
END_REGION

REGION Network 28: MM180 Z-Axis Screwdriver unit Clamps Open( QM180-MB180V - Q89.2 )
   RUNG wire#powerrail
      Contact( "Q_MM170_Z_Axis_Screwdrive_Unit_Downward_OP70_2" )
      wire#w1
      Contact( #Motion_Release )
      Coil( "Q_MM180_Z_Axis_Screwdrive_Unit_Clamps_Open_OP70_2" )
   END_RUNG
   RUNG wire#powerrail
      Contact( "Q_MM170_Z_Axis_Screwdrive_Unit_Upward_OP70_2" )
   END_RUNG wire#w1
   // the same network as SCL:
   "Q_MM180_Z_Axis_Screwdrive_Unit_Clamps_Open_OP70_2" := ("Q_MM170_Z_Axis_Screwdrive_Unit_Downward_OP70_2" OR "Q_MM170_Z_Axis_Screwdrive_Unit_Upward_OP70_2") AND #Motion_Release;
END_REGION

REGION Network 29: Hand line(36)
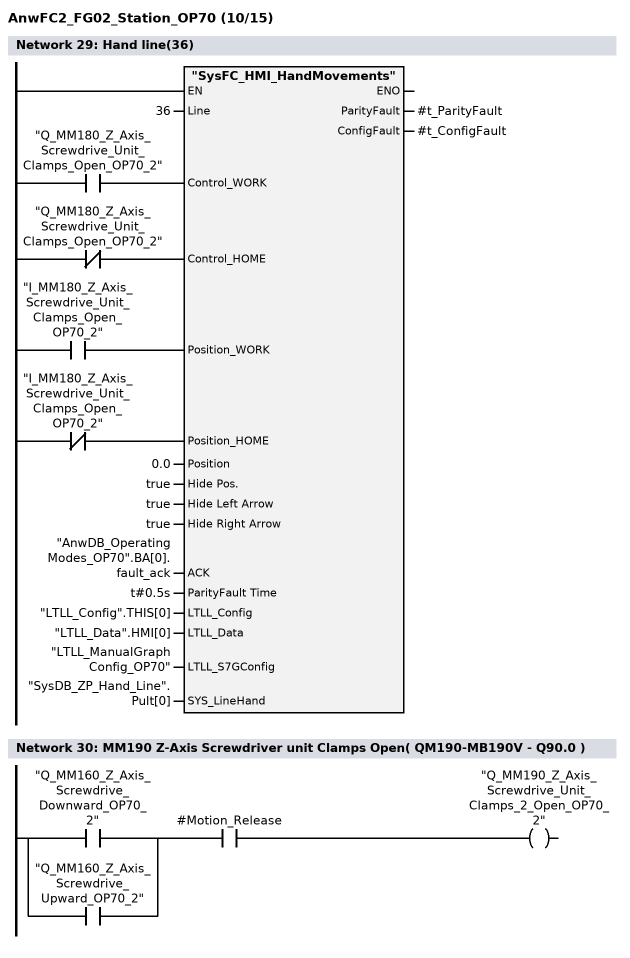
   RUNG wire#powerrail
      "SysFC_HMI_HandMovements"(Control_WORK := wire#w1, Control_HOME := wire#w2, Position_WORK := wire#w3, Position_HOME := wire#w4, Line := 36, Position := 0.0, "Hide Pos." := true, "Hide Left Arrow" := true, "Hide Right Arrow" := true, ACK := "AnwDB_OperatingModes_OP70".BA[0].fault_ack, "ParityFault Time" := t#0.5s, LTLL_Config := "LTLL_Config".THIS[0], LTLL_Data := "LTLL_Data".HMI[0], LTLL_S7GConfig := "LTLL_ManualGraphConfig_OP70", SYS_LineHand := "SysDB_ZP_Hand_Line".Pult[0], ParityFault => #t_ParityFault, ConfigFault => #t_ConfigFault)
   END_RUNG
   RUNG wire#powerrail
      Contact( "Q_MM180_Z_Axis_Screwdrive_Unit_Clamps_Open_OP70_2" )
   END_RUNG wire#w1
   RUNG wire#powerrail
      I_Contact( "Q_MM180_Z_Axis_Screwdrive_Unit_Clamps_Open_OP70_2" )
   END_RUNG wire#w2
   RUNG wire#powerrail
      Contact( "I_MM180_Z_Axis_Screwdrive_Unit_Clamps_Open_OP70_2" )
   END_RUNG wire#w3
   RUNG wire#powerrail
      I_Contact( "I_MM180_Z_Axis_Screwdrive_Unit_Clamps_Open_OP70_2" )
   END_RUNG wire#w4
   // the same network as SCL:
   "SysFC_HMI_HandMovements"(Line := 36,
                           Control_WORK := "Q_MM180_Z_Axis_Screwdrive_Unit_Clamps_Open_OP70_2",
                           Control_HOME := NOT "Q_MM180_Z_Axis_Screwdrive_Unit_Clamps_Open_OP70_2",
                           Position_WORK := "I_MM180_Z_Axis_Screwdrive_Unit_Clamps_Open_OP70_2",
                           Position_HOME := NOT "I_MM180_Z_Axis_Screwdrive_Unit_Clamps_Open_OP70_2",
                           Position := 0.0,
                           "Hide Pos." := true,
                           "Hide Left Arrow" := true,
                           "Hide Right Arrow" := true,
                           ACK := "AnwDB_OperatingModes_OP70".BA[0].fault_ack,
                           "ParityFault Time" := t#0.5s,
                           LTLL_Config := "LTLL_Config".THIS[0],
                           LTLL_Data := "LTLL_Data".HMI[0],
                           LTLL_S7GConfig := "LTLL_ManualGraphConfig_OP70",
                           SYS_LineHand := "SysDB_ZP_Hand_Line".Pult[0],
                           ParityFault => #t_ParityFault,
                           ConfigFault => #t_ConfigFault);
END_REGION

REGION Network 30: MM190 Z-Axis Screwdriver unit Clamps Open( QM190-MB190V - Q90.0 )
   RUNG wire#powerrail
      Contact( "Q_MM160_Z_Axis_Screwdrive_Downward_OP70_2" )
      wire#w1
      Contact( #Motion_Release )
      Coil( "Q_MM190_Z_Axis_Screwdrive_Unit_Clamps_2_Open_OP70_2" )
   END_RUNG
   RUNG wire#powerrail
      Contact( "Q_MM160_Z_Axis_Screwdrive_Upward_OP70_2" )
   END_RUNG wire#w1
   // the same network as SCL:
   "Q_MM190_Z_Axis_Screwdrive_Unit_Clamps_2_Open_OP70_2" := ("Q_MM160_Z_Axis_Screwdrive_Downward_OP70_2" OR "Q_MM160_Z_Axis_Screwdrive_Upward_OP70_2") AND #Motion_Release;
END_REGION

REGION Network 31: Hand line(37)
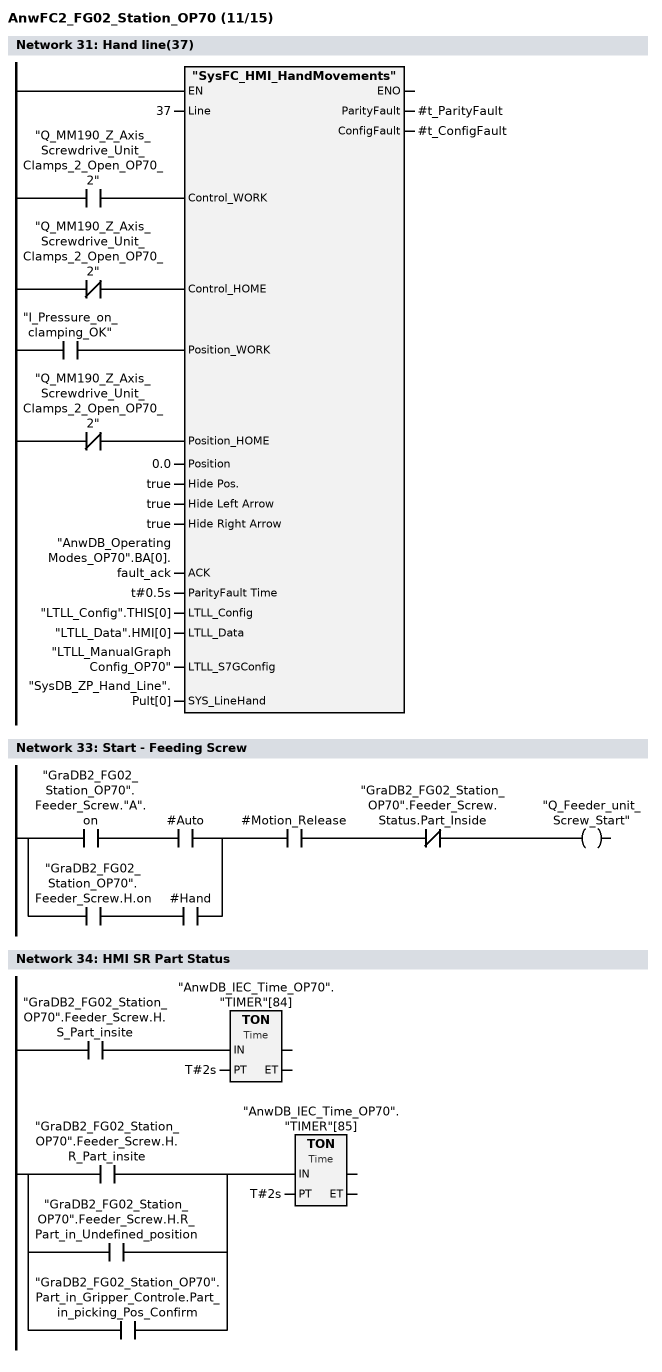
   RUNG wire#powerrail
      "SysFC_HMI_HandMovements"(Control_WORK := wire#w1, Control_HOME := wire#w2, Position_WORK := wire#w3, Position_HOME := wire#w4, Line := 37, Position := 0.0, "Hide Pos." := true, "Hide Left Arrow" := true, "Hide Right Arrow" := true, ACK := "AnwDB_OperatingModes_OP70".BA[0].fault_ack, "ParityFault Time" := t#0.5s, LTLL_Config := "LTLL_Config".THIS[0], LTLL_Data := "LTLL_Data".HMI[0], LTLL_S7GConfig := "LTLL_ManualGraphConfig_OP70", SYS_LineHand := "SysDB_ZP_Hand_Line".Pult[0], ParityFault => #t_ParityFault, ConfigFault => #t_ConfigFault)
   END_RUNG
   RUNG wire#powerrail
      Contact( "Q_MM190_Z_Axis_Screwdrive_Unit_Clamps_2_Open_OP70_2" )
   END_RUNG wire#w1
   RUNG wire#powerrail
      I_Contact( "Q_MM190_Z_Axis_Screwdrive_Unit_Clamps_2_Open_OP70_2" )
   END_RUNG wire#w2
   RUNG wire#powerrail
      Contact( "I_Pressure_on_clamping_OK" )
   END_RUNG wire#w3
   RUNG wire#powerrail
      I_Contact( "Q_MM190_Z_Axis_Screwdrive_Unit_Clamps_2_Open_OP70_2" )
   END_RUNG wire#w4
   // the same network as SCL:
   "SysFC_HMI_HandMovements"(Line := 37,
                           Control_WORK := "Q_MM190_Z_Axis_Screwdrive_Unit_Clamps_2_Open_OP70_2",
                           Control_HOME := NOT "Q_MM190_Z_Axis_Screwdrive_Unit_Clamps_2_Open_OP70_2",
                           Position_WORK := "I_Pressure_on_clamping_OK",
                           Position_HOME := NOT "Q_MM190_Z_Axis_Screwdrive_Unit_Clamps_2_Open_OP70_2",
                           Position := 0.0,
                           "Hide Pos." := true,
                           "Hide Left Arrow" := true,
                           "Hide Right Arrow" := true,
                           ACK := "AnwDB_OperatingModes_OP70".BA[0].fault_ack,
                           "ParityFault Time" := t#0.5s,
                           LTLL_Config := "LTLL_Config".THIS[0],
                           LTLL_Data := "LTLL_Data".HMI[0],
                           LTLL_S7GConfig := "LTLL_ManualGraphConfig_OP70",
                           SYS_LineHand := "SysDB_ZP_Hand_Line".Pult[0],
                           ParityFault => #t_ParityFault,
                           ConfigFault => #t_ConfigFault);
END_REGION

REGION Network 32: ################# FEEDING DEVICE #########################
END_REGION

REGION Network 33: Start - Feeding Screw
   RUNG wire#powerrail
      Contact( "GraDB2_FG02_Station_OP70".Feeder_Screw."A".on )
      Contact( #Auto )
      wire#w1
      Contact( #Motion_Release )
      I_Contact( "GraDB2_FG02_Station_OP70".Feeder_Screw.Status.Part_Inside )
      Coil( "Q_Feeder_unit_Screw_Start" )
   END_RUNG
   RUNG wire#powerrail
      Contact( "GraDB2_FG02_Station_OP70".Feeder_Screw.H.on )
      Contact( #Hand )
   END_RUNG wire#w1
   // the same network as SCL:
   "Q_Feeder_unit_Screw_Start" := (("GraDB2_FG02_Station_OP70".Feeder_Screw."A".on AND #Auto) OR ("GraDB2_FG02_Station_OP70".Feeder_Screw.H.on AND #Hand)) AND #Motion_Release AND NOT "GraDB2_FG02_Station_OP70".Feeder_Screw.Status.Part_Inside;
END_REGION

REGION Network 34: HMI SR Part Status
   RUNG wire#powerrail
      Contact( "GraDB2_FG02_Station_OP70".Feeder_Screw.H.S_Part_insite )
      { S7_Templates := "time_type := Time" } "AnwDB_IEC_Time_OP70"."TIMER"[84].TON(pt := T#2s, et =>)
   END_RUNG
   RUNG wire#powerrail
      Contact( "GraDB2_FG02_Station_OP70".Feeder_Screw.H.R_Part_insite )
      wire#w1
      { S7_Templates := "time_type := Time" } "AnwDB_IEC_Time_OP70"."TIMER"[85].TON(pt := T#2s, et =>)
   END_RUNG
   RUNG wire#powerrail
      Contact( "GraDB2_FG02_Station_OP70".Feeder_Screw.H.R_Part_in_Undefined_position )
   END_RUNG wire#w1
   RUNG wire#powerrail
      Contact( "GraDB2_FG02_Station_OP70".Part_in_Gripper_Controle.Part_in_picking_Pos_Confirm )
   END_RUNG wire#w1
   // the same network as SCL:
   "AnwDB_IEC_Time_OP70"."TIMER"[84].TON(IN := "GraDB2_FG02_Station_OP70".Feeder_Screw.H.S_Part_insite,
                           PT := T#2s);
   "AnwDB_IEC_Time_OP70"."TIMER"[85].TON(IN := "GraDB2_FG02_Station_OP70".Feeder_Screw.H.R_Part_insite OR "GraDB2_FG02_Station_OP70".Feeder_Screw.H.R_Part_in_Undefined_position OR "GraDB2_FG02_Station_OP70".Part_in_Gripper_Controle.Part_in_picking_Pos_Confirm,
                           PT := T#2s);
END_REGION

REGION Network 35: Part Inside
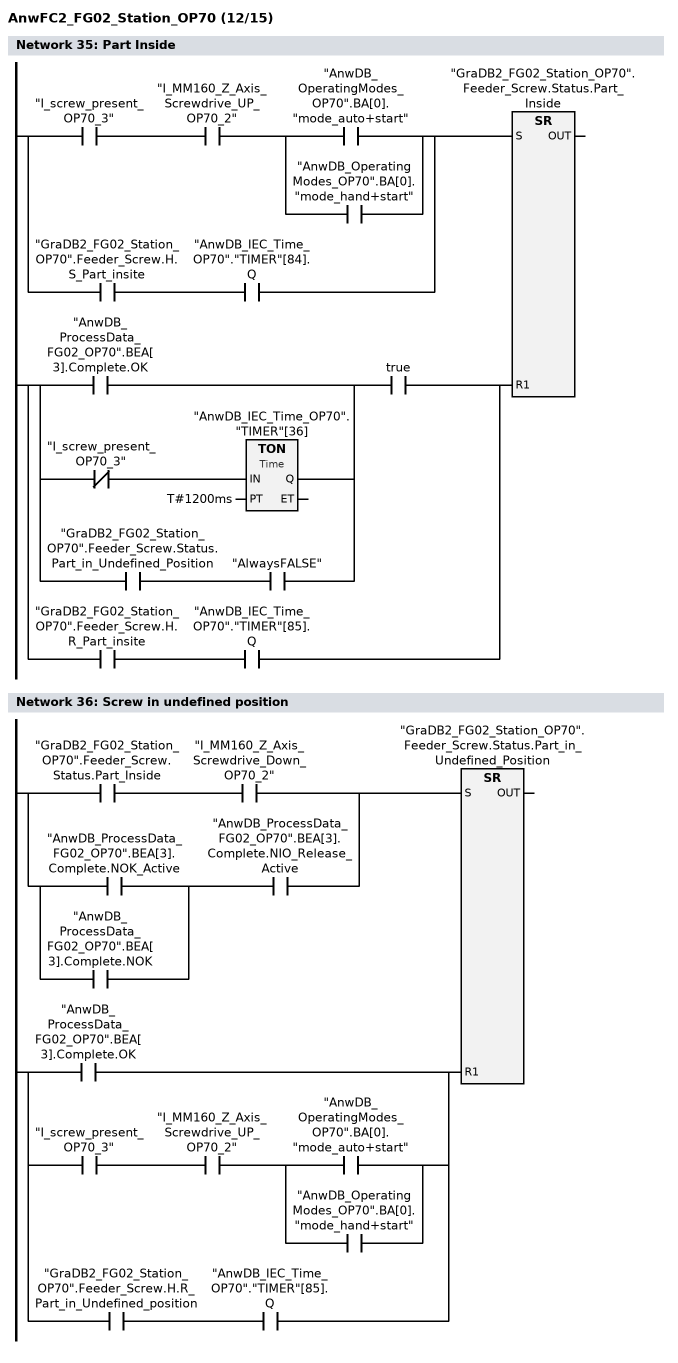
   RUNG wire#powerrail
      Contact( "I_screw_present_OP70_3" )
      Contact( "I_MM160_Z_Axis_Screwdrive_UP_OP70_2" )
      wire#w1
      Contact( "AnwDB_OperatingModes_OP70".BA[0]."mode_auto+start" )
      wire#w2
      S_SR(operand := "GraDB2_FG02_Station_OP70".Feeder_Screw.Status.Part_Inside, r1 := wire#w4)
   END_RUNG
   RUNG wire#w1
      Contact( "AnwDB_OperatingModes_OP70".BA[0]."mode_hand+start" )
   END_RUNG wire#w2
   RUNG wire#powerrail
      Contact( "GraDB2_FG02_Station_OP70".Feeder_Screw.H.S_Part_insite )
      Contact( "AnwDB_IEC_Time_OP70"."TIMER"[84].Q )
   END_RUNG wire#w2
   RUNG wire#powerrail
      Contact( "AnwDB_ProcessData_FG02_OP70".BEA[3].Complete.OK )
      wire#w3
      Contact( true )
   END_RUNG wire#w4
   RUNG wire#powerrail
      I_Contact( "I_screw_present_OP70_3" )
      { S7_Templates := "time_type := Time" } "AnwDB_IEC_Time_OP70"."TIMER"[36].TON(pt := T#1200ms, et =>)
   END_RUNG wire#w3
   RUNG wire#powerrail
      Contact( "GraDB2_FG02_Station_OP70".Feeder_Screw.Status.Part_in_Undefined_Position )
      Contact( "AlwaysFALSE" )
   END_RUNG wire#w3
   RUNG wire#powerrail
      Contact( "GraDB2_FG02_Station_OP70".Feeder_Screw.H.R_Part_insite )
      Contact( "AnwDB_IEC_Time_OP70"."TIMER"[85].Q )
   END_RUNG wire#w4
   // the same network as SCL:
   #_w1 := ("I_screw_present_OP70_3" AND "I_MM160_Z_Axis_Screwdrive_UP_OP70_2" AND ("AnwDB_OperatingModes_OP70".BA[0]."mode_auto+start" OR "AnwDB_OperatingModes_OP70".BA[0]."mode_hand+start")) OR ("GraDB2_FG02_Station_OP70".Feeder_Screw.H.S_Part_insite AND "AnwDB_IEC_Time_OP70"."TIMER"[84].Q);
   "AnwDB_IEC_Time_OP70"."TIMER"[36].TON(IN := NOT "I_screw_present_OP70_3", PT := T#1200ms);
   IF #_w1 THEN
       "GraDB2_FG02_Station_OP70".Feeder_Screw.Status.Part_Inside := TRUE;   // SR flip-flop
   END_IF;
   IF (("AnwDB_ProcessData_FG02_OP70".BEA[3].Complete.OK OR "AnwDB_IEC_Time_OP70"."TIMER"[36].Q OR ("GraDB2_FG02_Station_OP70".Feeder_Screw.Status.Part_in_Undefined_Position AND "AlwaysFALSE")) AND true) OR ("GraDB2_FG02_Station_OP70".Feeder_Screw.H.R_Part_insite AND "AnwDB_IEC_Time_OP70"."TIMER"[85].Q) THEN
       "GraDB2_FG02_Station_OP70".Feeder_Screw.Status.Part_Inside := FALSE;
   END_IF;
END_REGION

REGION Network 36: Screw in undefined position
   RUNG wire#powerrail
      Contact( "GraDB2_FG02_Station_OP70".Feeder_Screw.Status.Part_Inside )
      Contact( "I_MM160_Z_Axis_Screwdrive_Down_OP70_2" )
      wire#w1
      S_SR(operand := "GraDB2_FG02_Station_OP70".Feeder_Screw.Status.Part_in_Undefined_Position, r1 := wire#w4)
   END_RUNG
   RUNG wire#powerrail
      Contact( "AnwDB_ProcessData_FG02_OP70".BEA[3].Complete.NOK_Active )
      wire#w2
      Contact( "AnwDB_ProcessData_FG02_OP70".BEA[3].Complete.NIO_Release_Active )
   END_RUNG wire#w1
   RUNG wire#powerrail
      Contact( "AnwDB_ProcessData_FG02_OP70".BEA[3].Complete.NOK )
   END_RUNG wire#w2
   RUNG wire#powerrail
      Contact( "AnwDB_ProcessData_FG02_OP70".BEA[3].Complete.OK )
   END_RUNG wire#w4
   RUNG wire#powerrail
      Contact( "I_screw_present_OP70_3" )
      Contact( "I_MM160_Z_Axis_Screwdrive_UP_OP70_2" )
      wire#w3
      Contact( "AnwDB_OperatingModes_OP70".BA[0]."mode_auto+start" )
   END_RUNG wire#w4
   RUNG wire#w3
      Contact( "AnwDB_OperatingModes_OP70".BA[0]."mode_hand+start" )
   END_RUNG wire#w4
   RUNG wire#powerrail
      Contact( "GraDB2_FG02_Station_OP70".Feeder_Screw.H.R_Part_in_Undefined_position )
      Contact( "AnwDB_IEC_Time_OP70"."TIMER"[85].Q )
   END_RUNG wire#w4
   // the same network as SCL:
   IF ("GraDB2_FG02_Station_OP70".Feeder_Screw.Status.Part_Inside AND "I_MM160_Z_Axis_Screwdrive_Down_OP70_2") OR (("AnwDB_ProcessData_FG02_OP70".BEA[3].Complete.NOK_Active OR "AnwDB_ProcessData_FG02_OP70".BEA[3].Complete.NOK) AND "AnwDB_ProcessData_FG02_OP70".BEA[3].Complete.NIO_Release_Active) THEN
       "GraDB2_FG02_Station_OP70".Feeder_Screw.Status.Part_in_Undefined_Position := TRUE;   // SR flip-flop
   END_IF;
   IF "AnwDB_ProcessData_FG02_OP70".BEA[3].Complete.OK OR ("I_screw_present_OP70_3" AND "I_MM160_Z_Axis_Screwdrive_UP_OP70_2" AND ("AnwDB_OperatingModes_OP70".BA[0]."mode_auto+start" OR "AnwDB_OperatingModes_OP70".BA[0]."mode_hand+start")) OR ("GraDB2_FG02_Station_OP70".Feeder_Screw.H.R_Part_in_Undefined_position AND "AnwDB_IEC_Time_OP70"."TIMER"[85].Q) THEN
       "GraDB2_FG02_Station_OP70".Feeder_Screw.Status.Part_in_Undefined_Position := FALSE;
   END_IF;
END_REGION

REGION Network 37: ################# Gripper Status #########################
END_REGION

REGION Network 38: ################# PROCES STATUS #########################
END_REGION

REGION Network 39: BEA 2 - Ebit 1
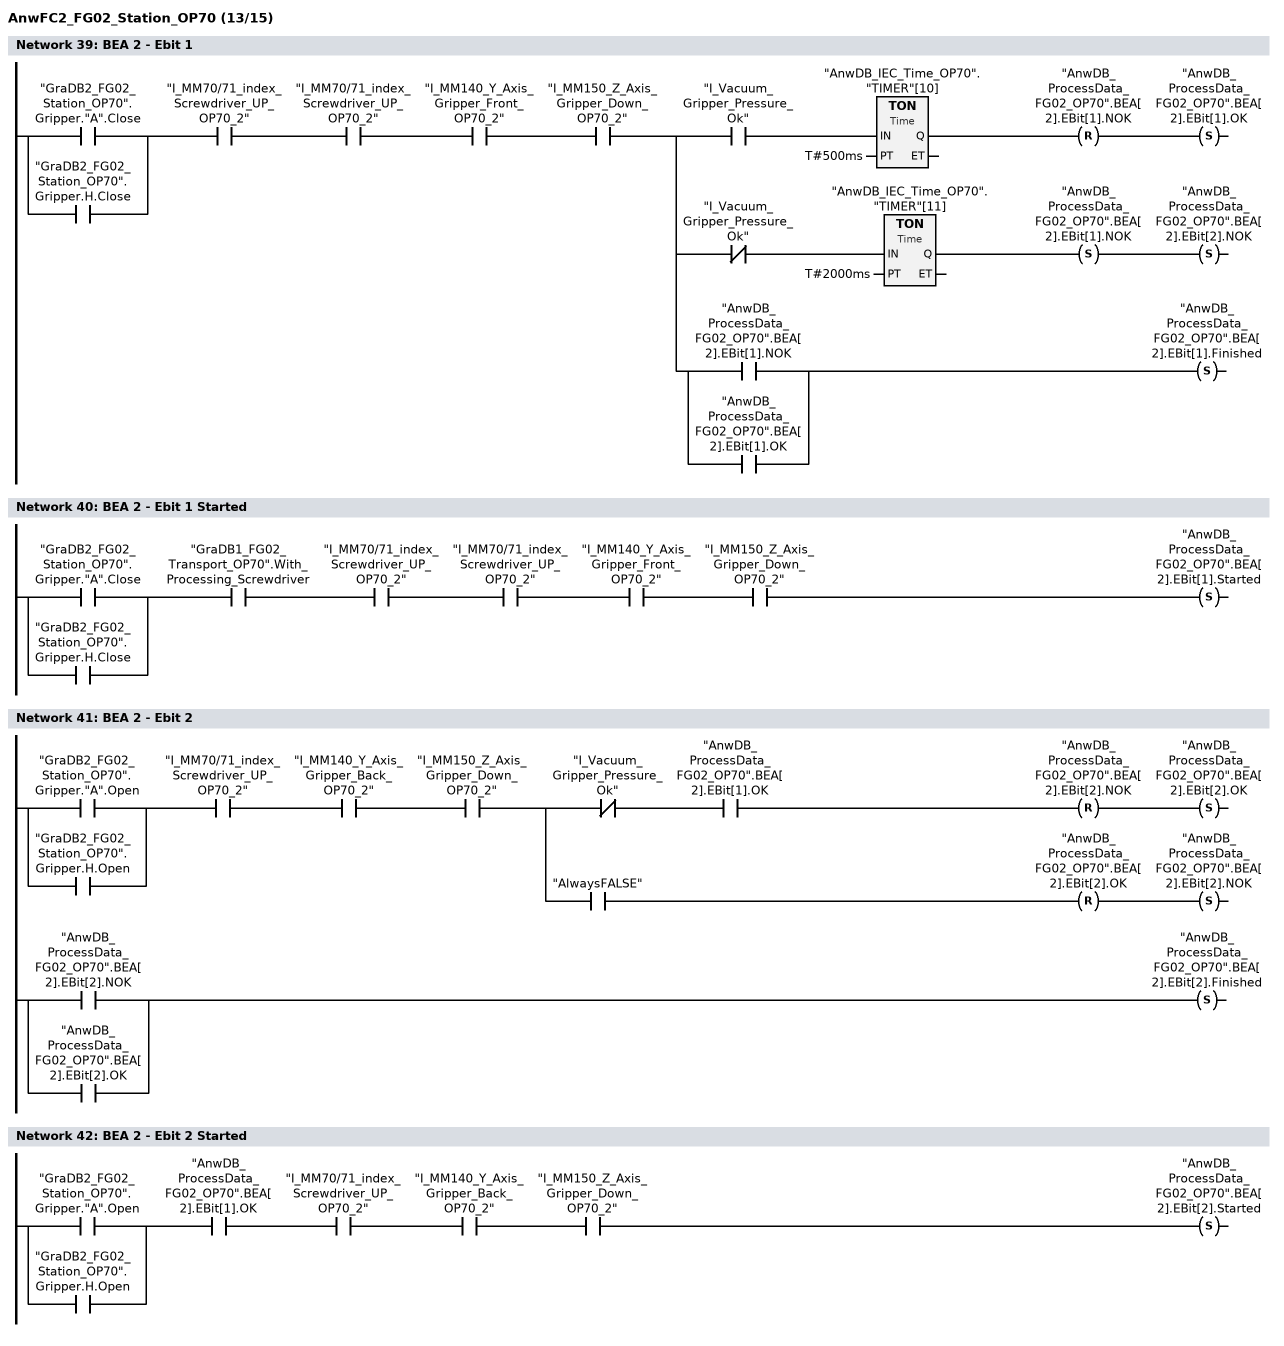
   RUNG wire#powerrail
      Contact( "GraDB2_FG02_Station_OP70".Gripper."A".Close )
      wire#w1
      Contact( "I_MM70/71_index_Screwdriver_UP_OP70_2" )
      Contact( "I_MM70/71_index_Screwdriver_UP_OP70_2" )
      Contact( "I_MM140_Y_Axis_Gripper_Front_OP70_2" )
      Contact( "I_MM150_Z_Axis_Gripper_Down_OP70_2" )
      wire#w2
      Contact( "I_Vacuum_Gripper_Pressure_Ok" )
      { S7_Templates := "time_type := Time" } "AnwDB_IEC_Time_OP70"."TIMER"[10].TON(pt := T#500ms, et =>)
      R_Coil( "AnwDB_ProcessData_FG02_OP70".BEA[2].EBit[1].NOK )
      S_Coil( "AnwDB_ProcessData_FG02_OP70".BEA[2].EBit[1].OK )
   END_RUNG
   RUNG wire#powerrail
      Contact( "GraDB2_FG02_Station_OP70".Gripper.H.Close )
   END_RUNG wire#w1
   RUNG wire#w2
      I_Contact( "I_Vacuum_Gripper_Pressure_Ok" )
      { S7_Templates := "time_type := Time" } "AnwDB_IEC_Time_OP70"."TIMER"[11].TON(pt := T#2000ms, et =>)
      S_Coil( "AnwDB_ProcessData_FG02_OP70".BEA[2].EBit[1].NOK )
      S_Coil( "AnwDB_ProcessData_FG02_OP70".BEA[2].EBit[2].NOK )
   END_RUNG
   RUNG wire#w2
      Contact( "AnwDB_ProcessData_FG02_OP70".BEA[2].EBit[1].NOK )
      wire#w3
      S_Coil( "AnwDB_ProcessData_FG02_OP70".BEA[2].EBit[1].Finished )
   END_RUNG
   RUNG wire#w2
      Contact( "AnwDB_ProcessData_FG02_OP70".BEA[2].EBit[1].OK )
   END_RUNG wire#w3
   // the same network as SCL:
   #_w1 := ("GraDB2_FG02_Station_OP70".Gripper."A".Close OR "GraDB2_FG02_Station_OP70".Gripper.H.Close) AND "I_MM70/71_index_Screwdriver_UP_OP70_2" AND "I_MM70/71_index_Screwdriver_UP_OP70_2" AND "I_MM140_Y_Axis_Gripper_Front_OP70_2" AND "I_MM150_Z_Axis_Gripper_Down_OP70_2";
   "AnwDB_IEC_Time_OP70"."TIMER"[10].TON(IN := #_w1 AND "I_Vacuum_Gripper_Pressure_Ok", PT := T#500ms);
   IF "AnwDB_IEC_Time_OP70"."TIMER"[10].Q THEN
       "AnwDB_ProcessData_FG02_OP70".BEA[2].EBit[1].NOK := FALSE;
       "AnwDB_ProcessData_FG02_OP70".BEA[2].EBit[1].OK := TRUE;
   END_IF;
   "AnwDB_IEC_Time_OP70"."TIMER"[11].TON(IN := #_w1 AND NOT "I_Vacuum_Gripper_Pressure_Ok", PT := T#2000ms);
   IF "AnwDB_IEC_Time_OP70"."TIMER"[11].Q THEN
       "AnwDB_ProcessData_FG02_OP70".BEA[2].EBit[1].NOK := TRUE;
       "AnwDB_ProcessData_FG02_OP70".BEA[2].EBit[2].NOK := TRUE;
   END_IF;
   IF #_w1 AND ("AnwDB_ProcessData_FG02_OP70".BEA[2].EBit[1].NOK OR "AnwDB_ProcessData_FG02_OP70".BEA[2].EBit[1].OK) THEN
       "AnwDB_ProcessData_FG02_OP70".BEA[2].EBit[1].Finished := TRUE;
   END_IF;
END_REGION

REGION Network 40: BEA 2 - Ebit 1 Started
   RUNG wire#powerrail
      Contact( "GraDB2_FG02_Station_OP70".Gripper."A".Close )
      wire#w1
      Contact( "GraDB1_FG02_Transport_OP70".With_Processing_Screwdriver )
      Contact( "I_MM70/71_index_Screwdriver_UP_OP70_2" )
      Contact( "I_MM70/71_index_Screwdriver_UP_OP70_2" )
      Contact( "I_MM140_Y_Axis_Gripper_Front_OP70_2" )
      Contact( "I_MM150_Z_Axis_Gripper_Down_OP70_2" )
      S_Coil( "AnwDB_ProcessData_FG02_OP70".BEA[2].EBit[1].Started )
   END_RUNG
   RUNG wire#powerrail
      Contact( "GraDB2_FG02_Station_OP70".Gripper.H.Close )
   END_RUNG wire#w1
   // the same network as SCL:
   IF ("GraDB2_FG02_Station_OP70".Gripper."A".Close OR "GraDB2_FG02_Station_OP70".Gripper.H.Close) AND "GraDB1_FG02_Transport_OP70".With_Processing_Screwdriver AND "I_MM70/71_index_Screwdriver_UP_OP70_2" AND "I_MM70/71_index_Screwdriver_UP_OP70_2" AND "I_MM140_Y_Axis_Gripper_Front_OP70_2" AND "I_MM150_Z_Axis_Gripper_Down_OP70_2" THEN
       "AnwDB_ProcessData_FG02_OP70".BEA[2].EBit[1].Started := TRUE;
   END_IF;
END_REGION

REGION Network 41: BEA 2 - Ebit 2
   RUNG wire#powerrail
      Contact( "GraDB2_FG02_Station_OP70".Gripper."A".Open )
      wire#w1
      Contact( "I_MM70/71_index_Screwdriver_UP_OP70_2" )
      Contact( "I_MM140_Y_Axis_Gripper_Back_OP70_2" )
      Contact( "I_MM150_Z_Axis_Gripper_Down_OP70_2" )
      wire#w2
      I_Contact( "I_Vacuum_Gripper_Pressure_Ok" )
      Contact( "AnwDB_ProcessData_FG02_OP70".BEA[2].EBit[1].OK )
      R_Coil( "AnwDB_ProcessData_FG02_OP70".BEA[2].EBit[2].NOK )
      S_Coil( "AnwDB_ProcessData_FG02_OP70".BEA[2].EBit[2].OK )
   END_RUNG
   RUNG wire#powerrail
      Contact( "GraDB2_FG02_Station_OP70".Gripper.H.Open )
   END_RUNG wire#w1
   RUNG wire#w2
      Contact( "AlwaysFALSE" )
      R_Coil( "AnwDB_ProcessData_FG02_OP70".BEA[2].EBit[2].OK )
      S_Coil( "AnwDB_ProcessData_FG02_OP70".BEA[2].EBit[2].NOK )
   END_RUNG
   RUNG wire#powerrail
      Contact( "AnwDB_ProcessData_FG02_OP70".BEA[2].EBit[2].NOK )
      wire#w3
      S_Coil( "AnwDB_ProcessData_FG02_OP70".BEA[2].EBit[2].Finished )
   END_RUNG
   RUNG wire#powerrail
      Contact( "AnwDB_ProcessData_FG02_OP70".BEA[2].EBit[2].OK )
   END_RUNG wire#w3
   // the same network as SCL:
   #_w1 := ("GraDB2_FG02_Station_OP70".Gripper."A".Open OR "GraDB2_FG02_Station_OP70".Gripper.H.Open) AND "I_MM70/71_index_Screwdriver_UP_OP70_2" AND "I_MM140_Y_Axis_Gripper_Back_OP70_2" AND "I_MM150_Z_Axis_Gripper_Down_OP70_2";
   #_w2 := #_w1 AND NOT "I_Vacuum_Gripper_Pressure_Ok" AND "AnwDB_ProcessData_FG02_OP70".BEA[2].EBit[1].OK;
   IF #_w2 THEN
       "AnwDB_ProcessData_FG02_OP70".BEA[2].EBit[2].NOK := FALSE;
       "AnwDB_ProcessData_FG02_OP70".BEA[2].EBit[2].OK := TRUE;
   END_IF;
   IF #_w1 AND "AlwaysFALSE" THEN
       "AnwDB_ProcessData_FG02_OP70".BEA[2].EBit[2].OK := FALSE;
       "AnwDB_ProcessData_FG02_OP70".BEA[2].EBit[2].NOK := TRUE;
   END_IF;
   IF "AnwDB_ProcessData_FG02_OP70".BEA[2].EBit[2].NOK OR "AnwDB_ProcessData_FG02_OP70".BEA[2].EBit[2].OK THEN
       "AnwDB_ProcessData_FG02_OP70".BEA[2].EBit[2].Finished := TRUE;
   END_IF;
END_REGION

REGION Network 42: BEA 2 - Ebit 2 Started
   RUNG wire#powerrail
      Contact( "GraDB2_FG02_Station_OP70".Gripper."A".Open )
      wire#w1
      Contact( "AnwDB_ProcessData_FG02_OP70".BEA[2].EBit[1].OK )
      Contact( "I_MM70/71_index_Screwdriver_UP_OP70_2" )
      Contact( "I_MM140_Y_Axis_Gripper_Back_OP70_2" )
      Contact( "I_MM150_Z_Axis_Gripper_Down_OP70_2" )
      S_Coil( "AnwDB_ProcessData_FG02_OP70".BEA[2].EBit[2].Started )
   END_RUNG
   RUNG wire#powerrail
      Contact( "GraDB2_FG02_Station_OP70".Gripper.H.Open )
   END_RUNG wire#w1
   // the same network as SCL:
   IF ("GraDB2_FG02_Station_OP70".Gripper."A".Open OR "GraDB2_FG02_Station_OP70".Gripper.H.Open) AND "AnwDB_ProcessData_FG02_OP70".BEA[2].EBit[1].OK AND "I_MM70/71_index_Screwdriver_UP_OP70_2" AND "I_MM140_Y_Axis_Gripper_Back_OP70_2" AND "I_MM150_Z_Axis_Gripper_Down_OP70_2" THEN
       "AnwDB_ProcessData_FG02_OP70".BEA[2].EBit[2].Started := TRUE;
   END_IF;
END_REGION

REGION Network 43: Part Fall Out
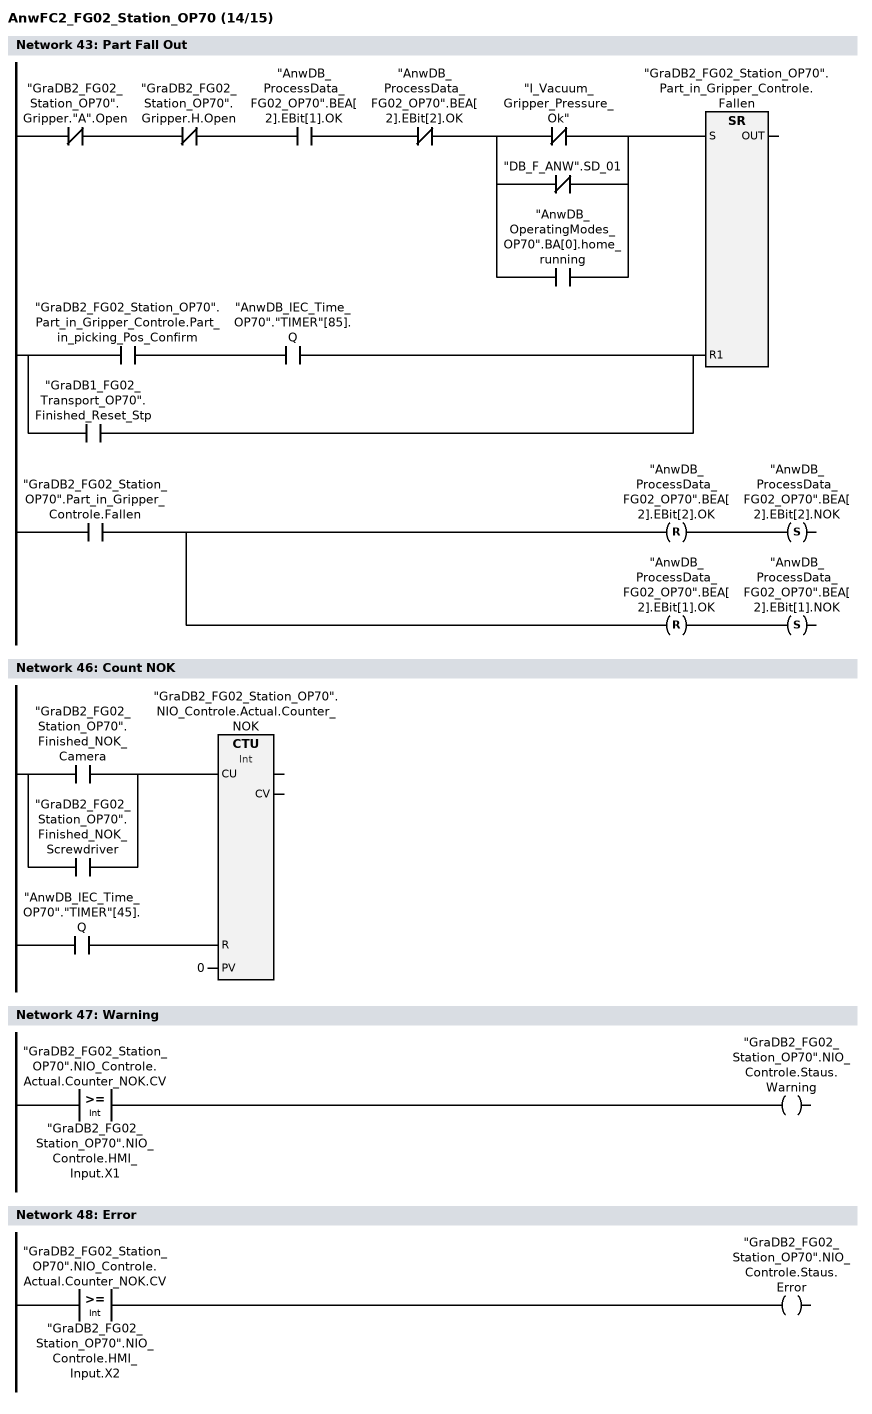
   RUNG wire#powerrail
      I_Contact( "GraDB2_FG02_Station_OP70".Gripper."A".Open )
      I_Contact( "GraDB2_FG02_Station_OP70".Gripper.H.Open )
      Contact( "AnwDB_ProcessData_FG02_OP70".BEA[2].EBit[1].OK )
      I_Contact( "AnwDB_ProcessData_FG02_OP70".BEA[2].EBit[2].OK )
      wire#w1
      I_Contact( "I_Vacuum_Gripper_Pressure_Ok" )
      wire#w2
      S_SR(operand := "GraDB2_FG02_Station_OP70".Part_in_Gripper_Controle.Fallen, r1 := wire#w3)
   END_RUNG
   RUNG wire#w1
      I_Contact( "DB_F_ANW".SD_01 )
   END_RUNG wire#w2
   RUNG wire#w1
      Contact( "AnwDB_OperatingModes_OP70".BA[0].home_running )
   END_RUNG wire#w2
   RUNG wire#powerrail
      Contact( "GraDB2_FG02_Station_OP70".Part_in_Gripper_Controle.Part_in_picking_Pos_Confirm )
      Contact( "AnwDB_IEC_Time_OP70"."TIMER"[85].Q )
   END_RUNG wire#w3
   RUNG wire#powerrail
      Contact( "GraDB1_FG02_Transport_OP70".Finished_Reset_Stp )
   END_RUNG wire#w3
   RUNG wire#powerrail
      Contact( "GraDB2_FG02_Station_OP70".Part_in_Gripper_Controle.Fallen )
      wire#w4
      R_Coil( "AnwDB_ProcessData_FG02_OP70".BEA[2].EBit[2].OK )
      S_Coil( "AnwDB_ProcessData_FG02_OP70".BEA[2].EBit[2].NOK )
   END_RUNG
   RUNG wire#w4
      R_Coil( "AnwDB_ProcessData_FG02_OP70".BEA[2].EBit[1].OK )
      S_Coil( "AnwDB_ProcessData_FG02_OP70".BEA[2].EBit[1].NOK )
   END_RUNG
   // the same network as SCL:
   IF NOT "GraDB2_FG02_Station_OP70".Gripper."A".Open AND NOT "GraDB2_FG02_Station_OP70".Gripper.H.Open AND "AnwDB_ProcessData_FG02_OP70".BEA[2].EBit[1].OK AND NOT "AnwDB_ProcessData_FG02_OP70".BEA[2].EBit[2].OK AND (NOT "I_Vacuum_Gripper_Pressure_Ok" OR NOT "DB_F_ANW".SD_01 OR "AnwDB_OperatingModes_OP70".BA[0].home_running) THEN
       "GraDB2_FG02_Station_OP70".Part_in_Gripper_Controle.Fallen := TRUE;   // SR flip-flop
   END_IF;
   IF ("GraDB2_FG02_Station_OP70".Part_in_Gripper_Controle.Part_in_picking_Pos_Confirm AND "AnwDB_IEC_Time_OP70"."TIMER"[85].Q) OR "GraDB1_FG02_Transport_OP70".Finished_Reset_Stp THEN
       "GraDB2_FG02_Station_OP70".Part_in_Gripper_Controle.Fallen := FALSE;
   END_IF;
   IF "GraDB2_FG02_Station_OP70".Part_in_Gripper_Controle.Fallen THEN
       "AnwDB_ProcessData_FG02_OP70".BEA[2].EBit[2].OK := FALSE;
       "AnwDB_ProcessData_FG02_OP70".BEA[2].EBit[2].NOK := TRUE;
       "AnwDB_ProcessData_FG02_OP70".BEA[2].EBit[1].OK := FALSE;
       "AnwDB_ProcessData_FG02_OP70".BEA[2].EBit[1].NOK := TRUE;
   END_IF;
END_REGION

REGION Network 44: ################ NIO Counting ################
END_REGION

REGION Network 45 (SCL): Rewrite Data from HMI
   #X1 := "GraDB2_FG02_Station_OP70".NIO_Controle.HMI_Input.X1;
   #X2 := "GraDB2_FG02_Station_OP70".NIO_Controle.HMI_Input.X2;


   REGION // Controle Input Data
       IF #X1 > #X2 THEN
           #X1 := "GraDB2_FG02_Station_OP70".NIO_Controle.HMI_Input.X1 := #X2;
       END_IF;
       IF #X1 <= 0 THEN
           #X1 := "GraDB2_FG02_Station_OP70".NIO_Controle.HMI_Input.X1 := 1;
       END_IF;

       IF #X2 <= 0 THEN
           #X2 := "GraDB2_FG02_Station_OP70".NIO_Controle.HMI_Input.X2 := 1;
       END_IF;
   END_REGION
END_REGION

REGION Network 46: Count NOK
   RUNG wire#powerrail
      Contact( "GraDB2_FG02_Station_OP70".Finished_NOK_Camera )
      wire#w1
      { S7_Templates := "value_type := Int" } "GraDB2_FG02_Station_OP70".NIO_Controle.Actual.Counter_NOK.CTU(r := wire#w2, pv := 0, cv =>)
   END_RUNG
   RUNG wire#powerrail
      Contact( "GraDB2_FG02_Station_OP70".Finished_NOK_Screwdriver )
   END_RUNG wire#w1
   RUNG wire#powerrail
      Contact( "AnwDB_IEC_Time_OP70"."TIMER"[45].Q )
   END_RUNG wire#w2
   // the same network as SCL:
   "GraDB2_FG02_Station_OP70".NIO_Controle.Actual.Counter_NOK.CTU(CU := "GraDB2_FG02_Station_OP70".Finished_NOK_Camera OR "GraDB2_FG02_Station_OP70".Finished_NOK_Screwdriver,
                           R := "AnwDB_IEC_Time_OP70"."TIMER"[45].Q,
                           PV := 0);
END_REGION

REGION Network 47: Warning
   RUNG wire#powerrail
      { S7_Templates := "SrcType := Int" } GE_Contact(in1 := "GraDB2_FG02_Station_OP70".NIO_Controle.Actual.Counter_NOK.CV, in2 := "GraDB2_FG02_Station_OP70".NIO_Controle.HMI_Input.X1)
      Coil( "GraDB2_FG02_Station_OP70".NIO_Controle.Staus.Warning )
   END_RUNG
   // the same network as SCL:
   "GraDB2_FG02_Station_OP70".NIO_Controle.Staus.Warning := "GraDB2_FG02_Station_OP70".NIO_Controle.Actual.Counter_NOK.CV >= "GraDB2_FG02_Station_OP70".NIO_Controle.HMI_Input.X1;
END_REGION

REGION Network 48: Error
   RUNG wire#powerrail
      { S7_Templates := "SrcType := Int" } GE_Contact(in1 := "GraDB2_FG02_Station_OP70".NIO_Controle.Actual.Counter_NOK.CV, in2 := "GraDB2_FG02_Station_OP70".NIO_Controle.HMI_Input.X2)
      Coil( "GraDB2_FG02_Station_OP70".NIO_Controle.Staus.Error )
   END_RUNG
   // the same network as SCL:
   "GraDB2_FG02_Station_OP70".NIO_Controle.Staus.Error := "GraDB2_FG02_Station_OP70".NIO_Controle.Actual.Counter_NOK.CV >= "GraDB2_FG02_Station_OP70".NIO_Controle.HMI_Input.X2;
END_REGION

REGION Network 49: ################ Number of Retry ################
END_REGION

REGION Network 50: Actual Number Of Retry - BEA 1
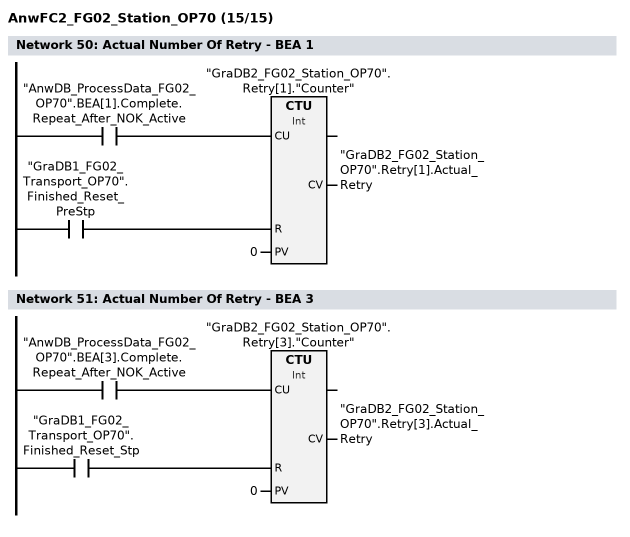
   RUNG wire#powerrail
      Contact( "AnwDB_ProcessData_FG02_OP70".BEA[1].Complete.Repeat_After_NOK_Active )
      { S7_Templates := "value_type := Int" } "GraDB2_FG02_Station_OP70".Retry[1]."Counter".CTU(r := wire#w1, pv := 0, cv => "GraDB2_FG02_Station_OP70".Retry[1].Actual_Retry)
   END_RUNG
   RUNG wire#powerrail
      Contact( "GraDB1_FG02_Transport_OP70".Finished_Reset_PreStp )
   END_RUNG wire#w1
   // the same network as SCL:
   "GraDB2_FG02_Station_OP70".Retry[1]."Counter".CTU(CU := "AnwDB_ProcessData_FG02_OP70".BEA[1].Complete.Repeat_After_NOK_Active,
                           R := "GraDB1_FG02_Transport_OP70".Finished_Reset_PreStp,
                           PV := 0,
                           CV => "GraDB2_FG02_Station_OP70".Retry[1].Actual_Retry);
END_REGION

REGION Network 51: Actual Number Of Retry - BEA 3
   RUNG wire#powerrail
      Contact( "AnwDB_ProcessData_FG02_OP70".BEA[3].Complete.Repeat_After_NOK_Active )
      { S7_Templates := "value_type := Int" } "GraDB2_FG02_Station_OP70".Retry[3]."Counter".CTU(r := wire#w1, pv := 0, cv => "GraDB2_FG02_Station_OP70".Retry[3].Actual_Retry)
   END_RUNG
   RUNG wire#powerrail
      Contact( "GraDB1_FG02_Transport_OP70".Finished_Reset_Stp )
   END_RUNG wire#w1
   // the same network as SCL:
   "GraDB2_FG02_Station_OP70".Retry[3]."Counter".CTU(CU := "AnwDB_ProcessData_FG02_OP70".BEA[3].Complete.Repeat_After_NOK_Active,
                           R := "GraDB1_FG02_Transport_OP70".Finished_Reset_Stp,
                           PV := 0,
                           CV => "GraDB2_FG02_Station_OP70".Retry[3].Actual_Retry);
END_REGION
END_FUNCTION
